C03626=1082.046,-23.655,-57.182,174.012,19.605,153.309
C03627=1082.052,-23.405,-57.194,174.013,19.607,153.309
C03628=1082.058,-23.155,-57.207,174.015,19.609,153.309
C03629=1082.064,-22.906,-57.220,174.016,19.611,153.310
C03630=1082.069,-22.656,-57.232,174.018,19.613,153.310
C03631=1082.075,-22.407,-57.246,174.019,19.615,153.310
C03632=1082.081,-22.157,-57.259,174.020,19.617,153.310
C03633=1082.087,-21.908,-57.272,174.022,19.619,153.310
C03634=1082.093,-21.658,-57.284,174.024,19.621,153.310
C03635=1082.099,-21.409,-57.298,174.025,19.623,153.310
C03636=1082.104,-21.158,-57.311,174.026,19.625,153.311
C03637=1082.110,-20.909,-57.324,174.028,19.627,153.311
C03638=1082.116,-20.659,-57.337,174.030,19.629,153.311
C03639=1082.122,-20.410,-57.350,174.031,19.631,153.311
C03640=1082.128,-20.160,-57.364,174.032,19.633,153.311
C03641=1082.134,-19.910,-57.376,174.034,19.635,153.311
C03642=1082.140,-19.661,-57.390,174.035,19.637,153.311
C03643=1082.146,-19.411,-57.402,174.037,19.639,153.311
C03644=1082.152,-19.162,-57.415,174.039,19.641,153.312
C03645=1082.157,-18.912,-57.429,174.040,19.643,153.312
C03646=1082.164,-18.663,-57.442,174.041,19.645,153.312
C03647=1082.170,-18.413,-57.455,174.042,19.647,153.312
C03648=1082.176,-18.163,-57.468,174.045,19.649,153.312
C03649=1082.181,-17.914,-57.482,174.046,19.651,153.312
C03650=1082.187,-17.664,-57.494,174.047,19.653,153.312
C03651=1082.194,-17.391,-57.509,174.048,19.655,153.313
C03652=1082.200,-17.116,-57.523,174.050,19.658,153.313
C03653=1082.206,-16.843,-57.538,174.052,19.660,153.313
C03654=1082.213,-16.568,-57.552,174.054,19.662,153.313
C03655=1082.220,-16.319,-57.565,174.055,19.664,153.313
C03656=1082.225,-16.069,-57.579,174.056,19.666,153.313
C03657=1082.231,-15.819,-57.592,174.058,19.668,153.313
C03658=1082.237,-15.570,-57.605,174.059,19.670,153.314
C03659=1082.243,-15.321,-57.618,174.061,19.672,153.314
C03660=1082.249,-15.071,-57.631,174.063,19.674,153.314
C03661=1082.255,-14.821,-57.645,174.064,19.676,153.314
C03662=1082.260,-14.572,-57.659,174.065,19.678,153.314
C03663=1082.266,-14.322,-57.671,174.066,19.680,153.314
C03664=1082.272,-14.073,-57.684,174.068,19.682,153.314
C03665=1082.278,-13.823,-57.698,174.070,19.684,153.314
C03666=1082.284,-13.574,-57.712,174.071,19.686,153.315
C03667=1082.289,-13.324,-57.725,174.072,19.688,153.315
C03668=1082.295,-13.074,-57.738,174.074,19.690,153.315
C03669=1082.301,-12.825,-57.752,174.076,19.692,153.315
C03670=1082.307,-12.576,-57.765,174.077,19.694,153.315
C03671=1082.312,-12.325,-57.778,174.078,19.696,153.315
C03672=1082.319,-12.076,-57.792,174.079,19.698,153.316
C03673=1082.324,-11.827,-57.805,174.082,19.700,153.316
C03674=1082.330,-11.577,-57.819,174.083,19.702,153.316
C03675=1082.336,-11.328,-57.833,174.084,19.704,153.316
C03676=1082.342,-11.078,-57.845,174.085,19.706,153.316
C03677=1082.348,-10.828,-57.859,174.087,19.708,153.316
C03678=1082.354,-10.578,-57.873,174.089,19.711,153.316
C03679=1082.360,-10.329,-57.886,174.090,19.713,153.317
C03680=1082.366,-10.079,-57.900,174.091,19.714,153.317
C03681=1082.372,-9.830,-57.913,174.093,19.716,153.317
C03682=1082.377,-9.580,-57.926,174.095,19.719,153.317
C03683=1082.383,-9.331,-57.939,174.096,19.721,153.317
C03684=1082.389,-9.081,-57.953,174.097,19.723,153.317
C03685=1082.395,-8.832,-57.967,174.099,19.725,153.318
C03686=1082.400,-8.582,-57.980,174.100,19.727,153.318
C03687=1082.407,-8.333,-57.994,174.102,19.729,153.318
C03688=1082.413,-8.083,-58.008,174.103,19.731,153.318
C03689=1082.418,-7.833,-58.022,174.105,19.733,153.318
C03690=1082.424,-7.584,-58.035,174.106,19.735,153.318
C03691=1082.430,-7.334,-58.048,174.108,19.738,153.318
C03692=1082.436,-7.084,-58.061,174.109,19.740,153.319
C03693=1082.441,-6.835,-58.075,174.110,19.742,153.319
C03694=1082.447,-6.586,-58.089,174.112,19.743,153.319
C03695=1082.454,-6.335,-58.103,174.113,19.745,153.319
C03696=1082.460,-6.086,-58.116,174.115,19.748,153.319
C03697=1082.465,-5.837,-58.130,174.117,19.750,153.319
C03698=1082.471,-5.587,-58.143,174.118,19.752,153.319
C03699=1082.477,-5.338,-58.157,174.119,19.754,153.320
C03700=1082.483,-5.088,-58.170,174.121,19.756,153.320
C03701=1082.489,-4.839,-58.184,174.123,19.758,153.320
C03702=1082.495,-4.589,-58.198,174.124,19.760,153.320
C03703=1082.501,-4.339,-58.212,174.125,19.762,153.320
C03704=1082.506,-4.090,-58.226,174.127,19.764,153.320
C03705=1082.513,-3.840,-58.239,174.128,19.766,153.320
C03706=1082.518,-3.591,-58.253,174.130,19.768,153.321
C03707=1082.525,-3.341,-58.266,174.131,19.770,153.321
C03708=1082.530,-3.091,-58.280,174.132,19.772,153.321
C03709=1082.536,-2.842,-58.294,174.134,19.775,153.321
C03710=1082.541,-2.592,-58.308,174.136,19.776,153.321
C03711=1082.548,-2.343,-58.321,174.137,19.778,153.321
C03712=1082.553,-2.094,-58.336,174.138,19.780,153.321
C03713=1082.559,-1.844,-58.350,174.140,19.783,153.322
C03714=1082.565,-1.594,-58.364,174.142,19.785,153.322
C03715=1082.571,-1.319,-58.379,174.143,19.787,153.322
C03716=1082.577,-1.043,-58.395,174.145,19.790,153.322
C03717=1082.584,-0.768,-58.409,174.146,19.792,153.322
C03718=1082.590,-0.492,-58.425,174.148,19.794,153.322
C03719=1082.596,-0.243,-58.439,174.149,19.796,153.323
C03720=1082.602,0.007,-58.452,174.151,19.798,153.323
C03721=1082.607,0.256,-58.466,174.153,19.801,153.323
C03722=1082.613,0.507,-58.480,174.154,19.803,153.323
C03723=1082.619,0.756,-58.494,174.155,19.805,153.323
C03724=1082.625,1.005,-58.508,174.156,19.807,153.323
C03725=1082.631,1.255,-58.522,174.158,19.809,153.324
C03726=1082.636,1.504,-58.536,174.160,19.811,153.324
C03727=1082.642,1.754,-58.550,174.161,19.813,153.324
C03728=1082.648,2.004,-58.564,174.162,19.815,153.324
C03729=1082.653,2.253,-58.579,174.164,19.818,153.324
C03730=1082.660,2.502,-58.592,174.166,19.820,153.324
C03731=1082.665,2.752,-58.606,174.167,19.821,153.324
C03732=1082.671,3.002,-58.620,174.168,19.823,153.325
C03733=1082.677,3.252,-58.634,174.170,19.826,153.325
C03734=1082.682,3.501,-58.649,174.172,19.828,153.325
C03735=1082.688,3.750,-58.662,174.173,19.830,153.325
C03736=1082.694,4.000,-58.677,174.174,19.832,153.325
C03737=1082.701,4.249,-58.691,174.176,19.834,153.325
C03738=1082.706,4.499,-58.704,174.178,19.836,153.326
C03739=1082.711,4.748,-58.718,174.179,19.838,153.326
C03740=1082.718,4.999,-58.733,174.180,19.840,153.326
C03741=1082.723,5.247,-58.747,174.182,19.843,153.326
C03742=1082.729,5.497,-58.761,174.183,19.845,153.326
C03743=1082.734,5.747,-58.775,174.185,19.847,153.326
C03744=1082.741,5.996,-58.790,174.186,19.849,153.327
C03745=1082.747,6.246,-58.803,174.188,19.851,153.327
C03746=1082.752,6.495,-58.817,174.189,19.853,153.327
C03747=1082.759,6.745,-58.832,174.190,19.855,153.327
C03748=1082.764,6.994,-58.846,174.192,19.857,153.327
C03749=1082.770,7.244,-58.860,174.194,19.859,153.327
C03750=1082.776,7.494,-58.875,174.195,19.861,153.327
C03751=1082.782,7.743,-58.888,174.197,19.863,153.328
C03752=1082.787,7.993,-58.902,174.199,19.866,153.328
C03753=1082.793,8.242,-58.917,174.200,19.868,153.328
C03754=1082.799,8.492,-58.931,174.201,19.870,153.328
C03755=1082.805,8.741,-58.945,174.202,19.872,153.328
C03756=1082.811,8.991,-58.959,174.205,19.874,153.328
C03757=1082.817,9.240,-58.974,174.206,19.876,153.329
C03758=1082.823,9.489,-58.988,174.207,19.878,153.329
C03759=1082.829,9.740,-59.002,174.208,19.880,153.329
C03760=1082.835,9.989,-59.017,174.210,19.883,153.329
C03761=1082.840,10.238,-59.030,174.212,19.884,153.329
C03762=1082.846,10.488,-59.045,174.213,19.886,153.329
C03763=1082.852,10.737,-59.059,174.214,19.888,153.330
C03764=1082.858,10.986,-59.074,174.217,19.891,153.330
C03765=1082.864,11.237,-59.088,174.218,19.893,153.330
C03766=1082.870,11.486,-59.103,174.219,19.895,153.330
C03767=1082.876,11.736,-59.117,174.221,19.897,153.330
C03768=1082.881,11.985,-59.131,174.222,19.899,153.330
C03769=1082.887,12.234,-59.145,174.224,19.902,153.330
C03770=1082.893,12.484,-59.160,174.225,19.904,153.331
C03771=1082.899,12.734,-59.174,174.227,19.906,153.331
C03772=1082.905,12.983,-59.189,174.228,19.907,153.331
C03773=1082.911,13.233,-59.203,174.230,19.909,153.331
C03774=1082.917,13.482,-59.217,174.231,19.911,153.331
C03775=1082.924,13.731,-59.232,174.233,19.914,153.331
C03776=1082.929,13.981,-59.246,174.234,19.916,153.332
C03777=1082.935,14.230,-59.261,174.236,19.918,153.332
C03778=1082.941,14.480,-59.275,174.238,19.920,153.332
C03779=1082.947,14.757,-59.291,174.239,19.922,153.332
C03780=1082.954,15.035,-59.307,174.241,19.925,153.332
C03781=1082.960,15.313,-59.323,174.242,19.927,153.332
C03782=1082.967,15.590,-59.339,174.244,19.930,153.333
C03783=1082.972,15.840,-59.354,174.245,19.932,153.333
C03784=1082.978,16.089,-59.369,174.247,19.934,153.333
C03785=1082.984,16.339,-59.384,174.249,19.936,153.333
C03786=1082.990,16.588,-59.398,174.250,19.938,153.333
C03787=1082.995,16.837,-59.412,174.252,19.940,153.333
C03788=1083.002,17.087,-59.427,174.253,19.942,153.333
C03789=1083.006,17.337,-59.442,174.255,19.944,153.334
C03790=1083.013,17.587,-59.457,174.256,19.946,153.334
C03791=1083.019,17.836,-59.471,174.257,19.948,153.334
C03792=1083.025,18.086,-59.485,174.260,19.951,153.334
C03793=1083.030,18.335,-59.500,174.261,19.953,153.334
C03794=1083.035,18.584,-59.515,174.262,19.955,153.334
C03795=1083.042,18.834,-59.529,174.263,19.957,153.335
C03796=1083.047,19.083,-59.544,174.265,19.959,153.335
C03797=1083.054,19.333,-59.559,174.267,19.961,153.335
C03798=1083.059,19.582,-59.574,174.268,19.963,153.335
C03799=1083.065,19.833,-59.588,174.270,19.966,153.335
C03800=1083.071,20.081,-59.603,174.271,19.968,153.335
C03801=1083.077,20.331,-59.618,174.273,19.970,153.336
C03802=1083.083,20.580,-59.632,174.275,19.972,153.336
C03803=1083.088,20.831,-59.647,174.276,19.974,153.336
C03804=1083.094,21.080,-59.662,174.277,19.976,153.336
C03805=1083.100,21.329,-59.676,174.278,19.978,153.336
C03806=1083.105,21.579,-59.692,174.281,19.981,153.336
C03807=1083.111,21.828,-59.707,174.282,19.983,153.337
C03808=1083.117,22.078,-59.721,174.283,19.985,153.337
C03809=1083.123,22.327,-59.735,174.285,19.987,153.337
C03810=1083.129,22.577,-59.751,174.286,19.989,153.337
C03811=1083.134,22.826,-59.765,174.288,19.991,153.337
C03812=1083.141,23.075,-59.780,174.290,19.993,153.337
C03813=1083.146,23.325,-59.796,174.291,19.995,153.337
C03814=1083.152,23.574,-59.811,174.293,19.997,153.338
C03815=1083.158,23.824,-59.824,174.294,19.999,153.338
C03816=1083.163,24.074,-59.840,174.296,20.002,153.338
C03817=1083.169,24.323,-59.855,174.297,20.004,153.338
C03818=1083.175,24.573,-59.870,174.298,20.006,153.338
C03819=1083.181,24.822,-59.885,174.301,20.008,153.338
C03820=1083.187,25.071,-59.900,174.302,20.010,153.339
C03821=1083.192,25.321,-59.915,174.303,20.012,153.339
C03822=1083.198,25.570,-59.930,174.305,20.015,153.339
C03823=1083.204,25.819,-59.944,174.306,20.017,153.339
C03824=1083.210,26.069,-59.960,174.308,20.019,153.339
C03825=1083.216,26.319,-59.975,174.310,20.021,153.339
C03826=1083.222,26.568,-59.989,174.311,20.023,153.340
C03827=1083.227,26.818,-60.004,174.312,20.025,153.340
C03828=1083.233,27.067,-60.019,174.315,20.028,153.340
C03829=1083.239,27.317,-60.034,174.316,20.030,153.340
C03830=1083.244,27.566,-60.049,174.317,20.031,153.340
C03831=1083.251,27.816,-60.064,174.319,20.033,153.340
C03832=1083.256,28.065,-60.079,174.321,20.036,153.340
C03833=1083.262,28.315,-60.094,174.322,20.038,153.341
C03834=1083.268,28.565,-60.109,174.323,20.040,153.341
C03835=1083.274,28.813,-60.125,174.325,20.042,153.341
C03836=1083.280,29.063,-60.140,174.327,20.044,153.341
C03837=1083.285,29.312,-60.155,174.328,20.046,153.341
C03838=1083.291,29.562,-60.170,174.330,20.049,153.341
C03839=1083.297,29.811,-60.185,174.331,20.051,153.342
C03840=1083.303,30.061,-60.201,174.332,20.053,153.342
C03841=1083.308,30.310,-60.215,174.335,20.055,153.342
C03842=1083.314,30.560,-60.231,174.336,20.057,153.342
C03843=1083.321,30.839,-60.247,174.338,20.060,153.342
C03844=1083.327,31.118,-60.265,174.339,20.062,153.342
C03845=1083.333,31.397,-60.281,174.341,20.065,153.343
C03846=1083.340,31.676,-60.299,174.342,20.067,153.343
C03847=1083.345,31.925,-60.313,174.344,20.069,153.343
C03848=1083.351,32.175,-60.330,174.346,20.071,153.343
C03849=1083.357,32.424,-60.344,174.347,20.073,153.343
C03850=1083.363,32.674,-60.360,174.349,20.076,153.343
C03851=1083.368,32.924,-60.375,174.351,20.077,153.343
C03852=1083.374,33.173,-60.390,174.352,20.079,153.344
C03853=1083.380,33.422,-60.405,174.354,20.082,153.344
C03854=1083.386,33.672,-60.420,174.355,20.084,153.344
C03855=1083.392,33.921,-60.436,174.357,20.086,153.344
C03856=1083.397,34.171,-60.452,174.359,20.088,153.344
C03857=1083.403,34.420,-60.466,174.360,20.090,153.344
C03858=1083.409,34.670,-60.482,174.361,20.092,153.345
C03859=1083.415,34.919,-60.498,174.363,20.095,153.345
C03860=1083.420,35.168,-60.513,174.365,20.097,153.345
C03861=1083.426,35.418,-60.528,174.366,20.099,153.345
C03862=1083.432,35.668,-60.543,174.368,20.101,153.345
C03863=1083.437,35.917,-60.558,174.369,20.103,153.345
C03864=1083.444,36.166,-60.574,174.371,20.105,153.345
C03865=1083.450,36.416,-60.590,174.373,20.107,153.346
C03866=1083.455,36.665,-60.605,174.374,20.109,153.346
C03867=1083.462,36.914,-60.620,174.375,20.111,153.346
C03868=1083.467,37.164,-60.636,174.377,20.113,153.346
C03869=1083.472,37.413,-60.651,174.379,20.115,153.346
C03870=1083.479,37.662,-60.667,174.380,20.117,153.346
C03871=1083.485,37.912,-60.682,174.382,20.120,153.347
C03872=1083.490,38.162,-60.698,174.383,20.122,153.347
C03873=1083.496,38.411,-60.712,174.385,20.124,153.347
C03874=1083.502,38.661,-60.729,174.387,20.126,153.347
C03875=1083.508,38.911,-60.744,174.388,20.128,153.347
C03876=1083.513,39.159,-60.760,174.390,20.131,153.347
C03877=1083.519,39.409,-60.776,174.392,20.132,153.347
C03878=1083.525,39.659,-60.791,174.393,20.134,153.348
C03879=1083.530,39.908,-60.806,174.395,20.137,153.348
C03880=1083.536,40.158,-60.822,174.396,20.139,153.348
C03881=1083.542,40.408,-60.838,174.398,20.141,153.348
C03882=1083.547,40.656,-60.853,174.400,20.143,153.348
C03883=1083.553,40.906,-60.868,174.401,20.145,153.348
C03884=1083.559,41.155,-60.885,174.402,20.147,153.349
C03885=1083.564,41.404,-60.900,174.404,20.150,153.349
C03886=1083.570,41.654,-60.916,174.406,20.152,153.349
C03887=1083.576,41.904,-60.932,174.407,20.154,153.349
C03888=1083.582,42.153,-60.947,174.409,20.156,153.349
C03889=1083.588,42.402,-60.962,174.410,20.158,153.349
C03890=1083.593,42.652,-60.978,174.412,20.161,153.350
C03891=1083.599,42.901,-60.994,174.414,20.162,153.350
C03892=1083.605,43.151,-61.010,174.415,20.164,153.350
C03893=1083.610,43.400,-61.026,174.417,20.167,153.350
C03894=1083.617,43.650,-61.041,174.419,20.169,153.350
C03895=1083.623,43.899,-61.057,174.420,20.171,153.350
C03896=1083.628,44.149,-61.072,174.422,20.173,153.350
C03897=1083.634,44.398,-61.088,174.423,20.175,153.351
C03898=1083.639,44.648,-61.104,174.424,20.177,153.351
C03899=1083.645,44.897,-61.120,174.427,20.180,153.351
C03900=1083.650,45.146,-61.135,174.428,20.182,153.351
C03901=1083.656,45.396,-61.152,174.430,20.184,153.351
C03902=1083.662,45.645,-61.168,174.431,20.186,153.351
C03903=1083.668,45.895,-61.183,174.433,20.188,153.352
C03904=1083.673,46.144,-61.199,174.435,20.190,153.352
C03905=1083.678,46.394,-61.215,174.436,20.192,153.352
C03906=1083.684,46.643,-61.232,174.437,20.194,153.352
C03907=1083.690,46.923,-61.249,174.439,20.197,153.352
C03908=1083.697,47.201,-61.267,174.441,20.199,153.352
C03909=1083.703,47.480,-61.285,174.443,20.201,153.353
C03910=1083.709,47.759,-61.302,174.445,20.204,153.353
C03911=1083.715,48.008,-61.319,174.446,20.206,153.353
C03912=1083.721,48.258,-61.335,174.448,20.208,153.353
C03913=1083.726,48.508,-61.350,174.450,20.210,153.353
C03914=1083.732,48.756,-61.366,174.452,20.213,153.353
C03915=1083.738,49.006,-61.382,174.453,20.215,153.353
C03916=1083.743,49.256,-61.398,174.454,20.217,153.354
C03917=1083.749,49.505,-61.414,174.456,20.219,153.354
C03918=1083.755,49.754,-61.431,174.458,20.221,153.354
C03919=1083.760,50.004,-61.446,174.460,20.224,153.354
C03920=1083.766,50.253,-61.462,174.461,20.225,153.354
C03921=1083.772,50.502,-61.478,174.462,20.227,153.354
C03922=1083.778,50.752,-61.494,174.465,20.230,153.354
C03923=1083.783,51.002,-61.511,174.466,20.232,153.355
C03924=1083.789,51.251,-61.527,174.467,20.234,153.355
C03925=1083.794,51.500,-61.543,174.469,20.236,153.355
C03926=1083.800,51.749,-61.559,174.471,20.238,153.355
C03927=1083.806,51.999,-61.575,174.473,20.240,153.355
C03928=1083.812,52.249,-61.591,174.474,20.242,153.355
C03929=1083.818,52.498,-61.607,174.475,20.244,153.356
C03930=1083.824,52.747,-61.623,174.478,20.246,153.356
C03931=1083.829,52.997,-61.639,174.479,20.248,153.356
C03932=1083.834,53.246,-61.655,174.481,20.251,153.356
C03933=1083.840,53.496,-61.672,174.482,20.253,153.356
C03934=1083.846,53.745,-61.688,174.484,20.255,153.356
C03935=1083.852,53.994,-61.704,174.486,20.257,153.356
C03936=1083.858,54.244,-61.720,174.487,20.259,153.356
C03937=1083.863,54.494,-61.736,174.489,20.261,153.357
C03938=1083.869,54.743,-61.752,174.491,20.263,153.357
C03939=1083.875,54.992,-61.768,174.492,20.265,153.357
C03940=1083.880,55.241,-61.785,174.494,20.268,153.357
C03941=1083.886,55.491,-61.801,174.495,20.269,153.357
C03942=1083.892,55.740,-61.817,174.498,20.272,153.357
C03943=1083.898,55.989,-61.834,174.499,20.274,153.357
C03944=1083.904,56.239,-61.850,174.500,20.276,153.358
C03945=1083.910,56.488,-61.866,174.502,20.278,153.358
C03946=1083.915,56.738,-61.882,174.504,20.280,153.358
C03947=1083.921,56.988,-61.899,174.506,20.282,153.358
C03948=1083.927,57.237,-61.915,174.507,20.284,153.358
C03949=1083.932,57.486,-61.931,174.508,20.286,153.358
C03950=1083.938,57.736,-61.947,174.511,20.288,153.358
C03951=1083.944,57.985,-61.964,174.512,20.290,153.359
C03952=1083.950,58.235,-61.980,174.514,20.292,153.359
C03953=1083.956,58.484,-61.997,174.516,20.294,153.359
C03954=1083.962,58.733,-62.013,174.517,20.296,153.359
C03955=1083.967,58.983,-62.029,174.519,20.298,153.359
C03956=1083.973,59.232,-62.046,174.520,20.300,153.359
C03957=1083.979,59.482,-62.062,174.523,20.303,153.359
C03958=1083.985,59.731,-62.079,174.524,20.305,153.360
C03959=1083.991,59.980,-62.095,174.525,20.306,153.360
C03960=1083.996,60.230,-62.111,174.527,20.309,153.360
C03961=1084.002,60.479,-62.128,174.529,20.311,153.360
C03962=1084.008,60.729,-62.144,174.531,20.313,153.360
C03963=1084.014,60.977,-62.161,174.532,20.315,153.360
C03964=1084.020,61.227,-62.177,174.534,20.317,153.360
C03965=1084.026,61.476,-62.194,174.536,20.319,153.360
C03966=1084.031,61.726,-62.211,174.537,20.321,153.360
C03967=1084.037,61.975,-62.227,174.539,20.323,153.361
C03968=1084.043,62.225,-62.243,174.541,20.325,153.361
C03969=1084.049,62.474,-62.259,174.543,20.327,153.361
C03970=1084.054,62.724,-62.276,174.544,20.329,153.361
C03971=1084.061,63.002,-62.295,174.546,20.331,153.361
C03972=1084.067,63.281,-62.313,174.548,20.333,153.361
C03973=1084.074,63.559,-62.331,174.550,20.336,153.361
C03974=1084.080,63.838,-62.349,174.552,20.338,153.362
C03975=1084.087,64.088,-62.367,174.554,20.340,153.362
C03976=1084.093,64.337,-62.384,174.556,20.342,153.362
C03977=1084.098,64.587,-62.400,174.557,20.344,153.362
C03978=1084.104,64.836,-62.417,174.558,20.346,153.362
C03979=1084.110,65.086,-62.433,174.561,20.348,153.362
C03980=1084.115,65.335,-62.450,174.562,20.350,153.362
C03981=1084.121,65.584,-62.467,174.564,20.353,153.362
C03982=1084.127,65.833,-62.483,174.565,20.354,153.362
C03983=1084.132,66.083,-62.500,174.568,20.356,153.363
C03984=1084.139,66.332,-62.517,174.569,20.358,153.363
C03985=1084.144,66.581,-62.534,174.571,20.361,153.363
C03986=1084.150,66.831,-62.550,174.573,20.362,153.363
C03987=1084.155,67.080,-62.567,174.574,20.364,153.363
C03988=1084.161,67.329,-62.584,174.576,20.367,153.363
C03989=1084.166,67.579,-62.601,174.577,20.369,153.363
C03990=1084.172,67.828,-62.617,174.580,20.371,153.363
C03991=1084.178,68.078,-62.634,174.581,20.373,153.364
C03992=1084.184,68.327,-62.651,174.583,20.375,153.364
C03993=1084.190,68.577,-62.668,174.585,20.377,153.364
C03994=1084.196,68.826,-62.684,174.586,20.379,153.364
C03995=1084.201,69.075,-62.702,174.588,20.381,153.364
C03996=1084.207,69.325,-62.718,174.589,20.383,153.364
C03997=1084.212,69.574,-62.735,174.592,20.385,153.364
C03998=1084.218,69.823,-62.752,174.593,20.387,153.364
C03999=1084.224,70.073,-62.769,174.595,20.389,153.365
C04000=1084.229,70.322,-62.786,174.596,20.391,153.365
C04001=1084.235,70.571,-62.802,174.599,20.393,153.365
C04002=1084.240,70.821,-62.819,174.600,20.395,153.365
C04003=1084.247,71.070,-62.837,174.601,20.397,153.365
C04004=1084.252,71.320,-62.854,174.604,20.399,153.365
C04005=1084.258,71.569,-62.871,174.605,20.401,153.365
C04006=1084.264,71.818,-62.887,174.607,20.404,153.365
C04007=1084.269,72.068,-62.904,174.608,20.405,153.366
C04008=1084.275,72.317,-62.922,174.611,20.408,153.366
C04009=1084.281,72.566,-62.938,174.612,20.410,153.366
C04010=1084.286,72.815,-62.956,174.614,20.412,153.366
C04011=1084.291,73.065,-62.972,174.616,20.414,153.366
C04012=1084.298,73.314,-62.990,174.618,20.416,153.366
C04013=1084.303,73.564,-63.007,174.619,20.417,153.366
C04014=1084.309,73.813,-63.024,174.620,20.419,153.366
C04015=1084.315,74.063,-63.040,174.623,20.422,153.367
C04016=1084.320,74.312,-63.058,174.624,20.423,153.367
C04017=1084.326,74.561,-63.075,174.626,20.426,153.367
C04018=1084.332,74.811,-63.092,174.628,20.428,153.367
C04019=1084.338,75.060,-63.109,174.630,20.430,153.367
C04020=1084.343,75.309,-63.127,174.631,20.432,153.367
C04021=1084.349,75.559,-63.143,174.633,20.434,153.367
C04022=1084.355,75.808,-63.160,174.635,20.436,153.367
C04023=1084.360,76.057,-63.178,174.637,20.438,153.367
C04024=1084.367,76.307,-63.195,174.638,20.440,153.368
C04025=1084.372,76.556,-63.212,174.641,20.442,153.368
C04026=1084.377,76.806,-63.229,174.642,20.444,153.368
C04027=1084.383,77.055,-63.247,174.643,20.445,153.368
C04028=1084.389,77.303,-63.264,174.646,20.448,153.368
C04029=1084.395,77.554,-63.281,174.647,20.450,153.368
C04030=1084.401,77.803,-63.298,174.649,20.452,153.368
C04031=1084.406,78.052,-63.315,174.650,20.454,153.368
C04032=1084.412,78.301,-63.332,174.653,20.456,153.368
C04033=1084.418,78.550,-63.350,174.654,20.458,153.368
C04034=1084.423,78.800,-63.367,174.656,20.460,153.369
C04035=1084.429,79.079,-63.386,174.658,20.463,153.369
C04036=1084.436,79.358,-63.406,174.660,20.464,153.369
C04037=1084.442,79.636,-63.425,174.662,20.467,153.369
C04038=1084.448,79.915,-63.445,174.664,20.469,153.369
C04039=1084.455,80.164,-63.462,174.665,20.471,153.369
C04040=1084.460,80.413,-63.480,174.668,20.473,153.369
C04041=1084.465,80.663,-63.496,174.669,20.475,153.369
C04042=1084.471,80.912,-63.514,174.671,20.477,153.370
C04043=1084.477,81.161,-63.532,174.673,20.479,153.370
C04044=1084.482,81.411,-63.549,174.675,20.481,153.370
C04045=1084.488,81.660,-63.566,174.676,20.483,153.370
C04046=1084.493,81.909,-63.584,174.679,20.485,153.370
C04047=1084.499,82.159,-63.602,174.680,20.487,153.370
C04048=1084.505,82.408,-63.619,174.682,20.489,153.370
C04049=1084.510,82.658,-63.636,174.684,20.491,153.370
C04050=1084.516,82.907,-63.654,174.686,20.493,153.370
C04051=1084.522,83.156,-63.672,174.687,20.495,153.371
C04052=1084.527,83.405,-63.689,174.689,20.497,153.371
C04053=1084.533,83.654,-63.706,174.691,20.499,153.371
C04054=1084.539,83.904,-63.723,174.693,20.501,153.371
C04055=1084.545,84.154,-63.741,174.694,20.503,153.371
C04056=1084.550,84.403,-63.759,174.697,20.505,153.371
C04057=1084.556,84.652,-63.776,174.698,20.507,153.371
C04058=1084.562,84.901,-63.794,174.700,20.509,153.371
C04059=1084.567,85.150,-63.812,174.702,20.511,153.371
C04060=1084.573,85.400,-63.829,174.704,20.513,153.371
C04061=1084.579,85.649,-63.847,174.705,20.515,153.372
C04062=1084.585,85.898,-63.865,174.708,20.517,153.372
C04063=1084.590,86.148,-63.882,174.709,20.519,153.372
C04064=1084.596,86.398,-63.900,174.711,20.521,153.372
C04065=1084.601,86.647,-63.917,174.713,20.523,153.372
C04066=1084.607,86.896,-63.935,174.715,20.525,153.372
C04067=1084.613,87.146,-63.953,174.716,20.527,153.372
C04068=1084.619,87.395,-63.970,174.719,20.529,153.372
C04069=1084.624,87.644,-63.988,174.720,20.531,153.372
C04070=1084.630,87.893,-64.006,174.722,20.533,153.372
C04071=1084.636,88.142,-64.023,174.724,20.535,153.373
C04072=1084.641,88.391,-64.041,174.726,20.537,153.373
C04073=1084.647,88.641,-64.059,174.727,20.538,153.373
C04074=1084.653,88.890,-64.076,174.730,20.540,153.373
C04075=1084.658,89.139,-64.094,174.731,20.542,153.373
C04076=1084.665,89.389,-64.112,174.733,20.544,153.373
C04077=1084.670,89.638,-64.129,174.735,20.546,153.373
C04078=1084.676,89.888,-64.147,174.737,20.548,153.373
C04079=1084.681,90.137,-64.165,174.738,20.550,153.373
C04080=1084.686,90.386,-64.183,174.741,20.552,153.373
C04081=1084.693,90.636,-64.201,174.742,20.554,153.373
C04082=1084.698,90.884,-64.219,174.744,20.556,153.373
C04083=1084.705,91.134,-64.237,174.746,20.558,153.373
C04084=1084.710,91.383,-64.255,174.748,20.560,153.374
C04085=1084.716,91.632,-64.272,174.749,20.561,153.374
C04086=1084.721,91.882,-64.291,174.751,20.564,153.374
C04087=1084.727,92.131,-64.308,174.753,20.565,153.374
C04088=1084.732,92.380,-64.326,174.755,20.568,153.374
C04089=1084.738,92.630,-64.344,174.757,20.569,153.374
C04090=1084.744,92.879,-64.362,174.759,20.572,153.374
C04091=1084.749,93.128,-64.381,174.760,20.573,153.374
C04092=1084.755,93.378,-64.398,174.762,20.576,153.374
C04093=1084.760,93.627,-64.416,174.765,20.577,153.374
C04094=1084.767,93.876,-64.434,174.766,20.579,153.375
C04095=1084.771,94.126,-64.452,174.768,20.581,153.375
C04096=1084.778,94.375,-64.471,174.770,20.583,153.375
C04097=1084.783,94.624,-64.488,174.772,20.585,153.375
C04098=1084.788,94.873,-64.506,174.774,20.587,153.375
C04099=1084.795,95.152,-64.526,174.776,20.589,153.375
C04100=1084.802,95.431,-64.547,174.778,20.592,153.375
C04101=1084.807,95.710,-64.567,174.780,20.594,153.375
C04102=1084.814,95.988,-64.587,174.782,20.596,153.375
C04103=1084.820,96.237,-64.605,174.784,20.597,153.375
C04104=1084.825,96.488,-64.623,174.786,20.600,153.375
C04105=1084.831,96.736,-64.642,174.788,20.601,153.375
C04106=1084.837,96.986,-64.659,174.790,20.603,153.375
C04107=1084.842,97.235,-64.677,174.791,20.605,153.376
C04108=1084.848,97.484,-64.696,174.794,20.607,153.376
C04109=1084.854,97.733,-64.714,174.795,20.609,153.376
C04110=1084.860,97.983,-64.732,174.797,20.611,153.376
C04111=1084.865,98.232,-64.751,174.799,20.613,153.376
C04112=1084.871,98.481,-64.769,174.801,20.615,153.376
C04113=1084.876,98.730,-64.786,174.803,20.616,153.376
C04114=1084.882,98.980,-64.805,174.805,20.618,153.376
C04115=1084.888,99.229,-64.823,174.807,20.621,153.376
C04116=1084.894,99.478,-64.842,174.809,20.622,153.376
C04117=1084.899,99.727,-64.860,174.811,20.624,153.376
C04118=1084.905,99.977,-64.878,174.812,20.626,153.376
C04119=1084.911,100.226,-64.896,174.815,20.628,153.376
C04120=1084.916,100.476,-64.915,174.816,20.630,153.377
C04121=1084.922,100.724,-64.933,174.818,20.632,153.377
C04122=1084.928,100.974,-64.951,174.820,20.633,153.377
C04123=1084.933,101.223,-64.969,174.822,20.635,153.377
C04124=1084.939,101.472,-64.988,174.824,20.638,153.377
C04125=1084.944,101.722,-65.006,174.826,20.639,153.377
C04126=1084.951,101.971,-65.024,174.828,20.641,153.377
C04127=1084.955,102.220,-65.043,174.830,20.643,153.377
C04128=1084.962,102.469,-65.061,174.832,20.645,153.377
C04129=1084.967,102.719,-65.079,174.833,20.647,153.377
C04130=1084.973,102.968,-65.098,174.836,20.649,153.377
C04131=1084.978,103.218,-65.117,174.838,20.651,153.377
C04132=1084.984,103.466,-65.135,174.839,20.652,153.377
C04133=1084.990,103.716,-65.153,174.842,20.655,153.377
C04134=1084.995,103.965,-65.172,174.843,20.656,153.378
C04135=1085.001,104.214,-65.191,174.845,20.659,153.378
C04136=1085.006,104.463,-65.209,174.847,20.660,153.378
C04137=1085.012,104.713,-65.228,174.849,20.662,153.378
C04138=1085.017,104.962,-65.246,174.852,20.664,153.378
C04139=1085.023,105.211,-65.264,174.853,20.666,153.378
C04140=1085.029,105.461,-65.283,174.855,20.668,153.378
C04141=1085.034,105.710,-65.302,174.857,20.669,153.378
C04142=1085.040,105.959,-65.321,174.859,20.672,153.378
C04143=1085.045,106.208,-65.339,174.860,20.673,153.378
C04144=1085.052,106.457,-65.357,174.863,20.675,153.378
C04145=1085.057,106.706,-65.376,174.865,20.678,153.378
C04146=1085.063,106.956,-65.394,174.866,20.679,153.378
C04147=1085.068,107.205,-65.413,174.869,20.681,153.378
C04148=1085.074,107.454,-65.432,174.870,20.682,153.378
C04149=1085.080,107.704,-65.450,174.872,20.685,153.379
C04150=1085.085,107.953,-65.469,174.874,20.686,153.379
C04151=1085.091,108.202,-65.488,174.876,20.688,153.379
C04152=1085.097,108.452,-65.506,174.879,20.690,153.379
C04153=1085.102,108.700,-65.525,174.880,20.692,153.379
C04154=1085.108,108.950,-65.544,174.882,20.694,153.379
C04155=1085.113,109.200,-65.562,174.884,20.696,153.379
C04156=1085.119,109.448,-65.581,174.886,20.698,153.379
C04157=1085.125,109.697,-65.600,174.889,20.699,153.379
C04158=1085.131,109.947,-65.619,174.890,20.701,153.379
C04159=1085.136,110.195,-65.637,174.892,20.703,153.379
C04160=1085.142,110.445,-65.656,174.894,20.705,153.379
C04161=1085.148,110.695,-65.675,174.896,20.707,153.379
C04162=1085.153,110.943,-65.693,174.899,20.709,153.379
C04163=1085.160,111.222,-65.715,174.900,20.711,153.379
C04164=1085.166,111.501,-65.736,174.902,20.713,153.379
C04165=1085.172,111.780,-65.757,174.905,20.714,153.379
C04166=1085.178,112.059,-65.778,174.907,20.717,153.379
C04167=1085.184,112.308,-65.797,174.909,20.719,153.379
C04168=1085.190,112.557,-65.816,174.911,20.720,153.379
C04169=1085.196,112.806,-65.835,174.913,20.722,153.379
C04170=1085.201,113.056,-65.854,174.915,20.724,153.380
C04171=1085.207,113.306,-65.872,174.917,20.726,153.380
C04172=1085.212,113.554,-65.891,174.919,20.728,153.380
C04173=1085.218,113.803,-65.910,174.921,20.729,153.380
C04174=1085.224,114.053,-65.929,174.923,20.731,153.380
C04175=1085.229,114.302,-65.948,174.925,20.733,153.380
C04176=1085.235,114.551,-65.967,174.927,20.735,153.380
C04177=1085.241,114.800,-65.986,174.929,20.737,153.380
C04178=1085.247,115.050,-66.005,174.931,20.739,153.380
C04179=1085.252,115.298,-66.024,174.933,20.741,153.380
C04180=1085.257,115.548,-66.043,174.935,20.742,153.380
C04181=1085.263,115.797,-66.062,174.937,20.744,153.380
C04182=1085.268,116.046,-66.081,174.939,20.746,153.380
C04183=1085.274,116.295,-66.101,174.941,20.748,153.380
C04184=1085.280,116.545,-66.120,174.943,20.750,153.380
C04185=1085.285,116.794,-66.139,174.945,20.752,153.380
C04186=1085.290,117.043,-66.158,174.947,20.754,153.380
C04187=1085.296,117.292,-66.177,174.949,20.756,153.380
C04188=1085.302,117.542,-66.196,174.951,20.757,153.380
C04189=1085.307,117.791,-66.215,174.953,20.759,153.381
C04190=1085.313,118.040,-66.235,174.955,20.761,153.381
C04191=1085.318,118.289,-66.254,174.957,20.763,153.381
C04192=1085.323,118.538,-66.273,174.959,20.765,153.381
C04193=1085.329,118.788,-66.292,174.961,20.767,153.381
C04194=1085.335,119.037,-66.311,174.964,20.769,153.381
C04195=1085.340,119.286,-66.330,174.965,20.770,153.381
C04196=1085.345,119.535,-66.349,174.968,20.772,153.381
C04197=1085.351,119.784,-66.369,174.970,20.774,153.381
C04198=1085.357,120.033,-66.389,174.971,20.776,153.381
C04199=1085.363,120.283,-66.408,174.974,20.778,153.381
C04200=1085.368,120.532,-66.427,174.975,20.779,153.381
C04201=1085.374,120.781,-66.446,174.978,20.781,153.381
C04202=1085.379,121.030,-66.465,174.980,20.783,153.381
C04203=1085.385,121.280,-66.484,174.981,20.784,153.381
C04204=1085.391,121.529,-66.504,174.984,20.786,153.381
C04205=1085.396,121.777,-66.523,174.986,20.788,153.381
C04206=1085.402,122.027,-66.542,174.988,20.790,153.381
C04207=1085.407,122.276,-66.562,174.990,20.792,153.381
C04208=1085.413,122.525,-66.582,174.992,20.794,153.381
C04209=1085.419,122.775,-66.601,174.994,20.796,153.381
C04210=1085.424,123.024,-66.621,174.996,20.797,153.381
C04211=1085.429,123.273,-66.640,174.999,20.799,153.381
C04212=1085.435,123.522,-66.660,175.000,20.801,153.381
C04213=1085.441,123.771,-66.679,175.002,20.803,153.381
C04214=1085.447,124.021,-66.698,175.005,20.805,153.381
C04215=1085.452,124.270,-66.717,175.006,20.806,153.382
C04216=1085.458,124.519,-66.737,175.009,20.808,153.382
C04217=1085.464,124.768,-66.756,175.011,20.810,153.382
C04218=1085.469,125.017,-66.775,175.013,20.811,153.382
C04219=1085.475,125.266,-66.795,175.015,20.813,153.382
C04220=1085.481,125.515,-66.815,175.017,20.815,153.382
C04221=1085.486,125.765,-66.834,175.019,20.817,153.382
C04222=1085.492,126.014,-66.854,175.021,20.819,153.382
C04223=1085.497,126.263,-66.874,175.024,20.821,153.382
C04224=1085.503,126.513,-66.893,175.025,20.822,153.382
C04225=1085.509,126.762,-66.913,175.028,20.824,153.382
C04226=1085.515,127.011,-66.932,175.030,20.826,153.382
C04227=1085.521,127.289,-66.954,175.032,20.828,153.382
C04228=1085.527,127.568,-66.976,175.034,20.829,153.382
C04229=1085.533,127.847,-66.997,175.036,20.831,153.382
C04230=1085.540,128.126,-67.020,175.039,20.833,153.382
C04231=1085.545,128.376,-67.039,175.041,20.835,153.382
C04232=1085.551,128.624,-67.059,175.043,20.837,153.382
C04233=1085.557,128.874,-67.079,175.046,20.839,153.382
C04234=1085.563,129.123,-67.099,175.047,20.840,153.382
C04235=1085.568,129.371,-67.117,175.050,20.842,153.382
C04236=1085.574,129.620,-67.137,175.052,20.844,153.382
C04237=1085.579,129.870,-67.157,175.054,20.845,153.382
C04238=1085.585,130.119,-67.177,175.056,20.847,153.382
C04239=1085.591,130.368,-67.196,175.059,20.849,153.382
C04240=1085.597,130.617,-67.216,175.060,20.850,153.382
C04241=1085.602,130.866,-67.236,175.062,20.852,153.382
C04242=1085.608,131.115,-67.256,175.065,20.854,153.382
C04243=1085.614,131.364,-67.276,175.067,20.855,153.382
C04244=1085.619,131.614,-67.295,175.069,20.857,153.382
C04245=1085.625,131.863,-67.315,175.071,20.859,153.382
C04246=1085.631,132.112,-67.335,175.073,20.860,153.382
C04247=1085.636,132.361,-67.355,175.075,20.862,153.382
C04248=1085.642,132.611,-67.374,175.078,20.864,153.382
C04249=1085.648,132.859,-67.394,175.080,20.866,153.382
C04250=1085.653,133.109,-67.415,175.082,20.868,153.382
C04251=1085.659,133.358,-67.434,175.084,20.870,153.382
C04252=1085.665,133.607,-67.454,175.087,20.871,153.382
C04253=1085.670,133.856,-67.475,175.088,20.872,153.382
C04254=1085.676,134.105,-67.494,175.090,20.874,153.382
C04255=1085.681,134.354,-67.514,175.093,20.876,153.382
C04256=1085.687,134.603,-67.534,175.094,20.878,153.382
C04257=1085.693,134.853,-67.554,175.097,20.880,153.382
C04258=1085.698,135.102,-67.574,175.099,20.881,153.382
C04259=1085.704,135.351,-67.594,175.101,20.883,153.382
C04260=1085.709,135.600,-67.614,175.103,20.885,153.382
C04261=1085.715,135.849,-67.634,175.106,20.886,153.382
C04262=1085.720,136.098,-67.655,175.108,20.888,153.382
C04263=1085.726,136.347,-67.674,175.110,20.890,153.382
C04264=1085.732,136.597,-67.694,175.112,20.892,153.382
C04265=1085.738,136.846,-67.715,175.114,20.893,153.382
C04266=1085.744,137.095,-67.735,175.117,20.895,153.382
C04267=1085.749,137.344,-67.755,175.118,20.897,153.382
C04268=1085.755,137.593,-67.775,175.121,20.898,153.382
C04269=1085.760,137.843,-67.795,175.123,20.900,153.382
C04270=1085.766,138.092,-67.815,175.126,20.902,153.382
C04271=1085.771,138.341,-67.835,175.127,20.903,153.382
C04272=1085.777,138.590,-67.855,175.129,20.905,153.382
C04273=1085.783,138.839,-67.876,175.132,20.907,153.382
C04274=1085.789,139.088,-67.896,175.134,20.908,153.382
C04275=1085.793,139.337,-67.916,175.136,20.910,153.382
C04276=1085.799,139.586,-67.936,175.138,20.912,153.382
C04277=1085.805,139.835,-67.956,175.141,20.914,153.382
C04278=1085.811,140.085,-67.977,175.142,20.915,153.382
C04279=1085.817,140.334,-67.997,175.145,20.917,153.382
C04280=1085.823,140.583,-68.017,175.147,20.919,153.382
C04281=1085.828,140.832,-68.038,175.150,20.921,153.382
C04282=1085.833,141.081,-68.058,175.151,20.922,153.382
C04283=1085.839,141.330,-68.078,175.154,20.924,153.382
C04284=1085.844,141.579,-68.099,175.156,20.925,153.382
C04285=1085.850,141.828,-68.119,175.159,20.927,153.382
C04286=1085.856,142.077,-68.139,175.160,20.929,153.382
C04287=1085.861,142.327,-68.159,175.162,20.931,153.382
C04288=1085.866,142.576,-68.180,175.165,20.933,153.382
C04289=1085.872,142.825,-68.200,175.167,20.934,153.382
C04290=1085.878,143.074,-68.221,175.169,20.936,153.382
C04291=1085.884,143.352,-68.244,175.171,20.937,153.382
C04292=1085.890,143.632,-68.266,175.175,20.940,153.382
C04293=1085.896,143.910,-68.290,175.177,20.942,153.382
C04294=1085.903,144.189,-68.312,175.179,20.944,153.382
C04295=1085.909,144.438,-68.332,175.182,20.945,153.382
C04296=1085.914,144.687,-68.353,175.183,20.946,153.382
C04297=1085.919,144.936,-68.373,175.186,20.948,153.382
C04298=1085.924,145.185,-68.394,175.188,20.950,153.382
C04299=1085.931,145.433,-68.415,175.191,20.952,153.382
C04300=1085.937,145.683,-68.436,175.192,20.953,153.382
C04301=1085.942,145.932,-68.456,175.195,20.955,153.382
C04302=1085.948,146.181,-68.476,175.197,20.956,153.382
C04303=1085.953,146.430,-68.497,175.200,20.958,153.382
C04304=1085.958,146.679,-68.517,175.201,20.960,153.382
C04305=1085.965,146.929,-68.537,175.204,20.961,153.382
C04306=1085.971,147.177,-68.559,175.206,20.963,153.382
C04307=1085.976,147.426,-68.579,175.209,20.965,153.382
C04308=1085.981,147.676,-68.600,175.211,20.966,153.381
C04309=1085.988,147.925,-68.620,175.213,20.968,153.382
C04310=1085.993,148.174,-68.641,175.215,20.970,153.382
C04311=1085.998,148.423,-68.662,175.218,20.971,153.381
C04312=1086.004,148.672,-68.683,175.220,20.973,153.381
C04313=1086.009,148.921,-68.703,175.222,20.975,153.381
C04314=1086.015,149.171,-68.724,175.224,20.977,153.381
C04315=1086.021,149.419,-68.745,175.227,20.978,153.381
C04316=1086.026,149.668,-68.765,175.229,20.980,153.381
C04317=1086.032,149.917,-68.786,175.231,20.982,153.381
C04318=1086.037,150.167,-68.807,175.233,20.983,153.381
C04319=1086.043,150.416,-68.828,175.236,20.985,153.381
C04320=1086.048,150.665,-68.849,175.238,20.987,153.381
C04321=1086.054,150.914,-68.869,175.241,20.988,153.381
C04322=1086.060,151.163,-68.891,175.243,20.990,153.381
C04323=1086.066,151.412,-68.911,175.244,20.991,153.381
C04324=1086.071,151.661,-68.931,175.247,20.993,153.381
C04325=1086.077,151.909,-68.953,175.249,20.995,153.381
C04326=1086.082,152.159,-68.973,175.252,20.996,153.381
C04327=1086.088,152.408,-68.994,175.254,20.998,153.381
C04328=1086.093,152.657,-69.015,175.256,20.999,153.381
C04329=1086.098,152.906,-69.036,175.258,21.001,153.381
C04330=1086.105,153.155,-69.057,175.261,21.003,153.381
C04331=1086.110,153.404,-69.078,175.263,21.005,153.381
C04332=1086.115,153.654,-69.099,175.266,21.006,153.381
C04333=1086.121,153.903,-69.120,175.267,21.007,153.381
C04334=1086.127,154.152,-69.141,175.270,21.009,153.381
C04335=1086.132,154.400,-69.162,175.272,21.011,153.381
C04336=1086.138,154.650,-69.183,175.275,21.013,153.381
C04337=1086.144,154.899,-69.204,175.277,21.015,153.381
C04338=1086.149,155.148,-69.225,175.280,21.016,153.381
C04339=1086.155,155.397,-69.246,175.281,21.017,153.381
C04340=1086.160,155.646,-69.267,175.284,21.019,153.381
C04341=1086.166,155.895,-69.288,175.286,21.021,153.381
C04342=1086.172,156.144,-69.309,175.289,21.023,153.381
C04343=1086.177,156.393,-69.330,175.291,21.024,153.381
C04344=1086.182,156.642,-69.351,175.294,21.026,153.381
C04345=1086.189,156.891,-69.373,175.295,21.027,153.381
C04346=1086.194,157.140,-69.393,175.298,21.029,153.381
C04347=1086.199,157.389,-69.414,175.300,21.031,153.381
C04348=1086.206,157.638,-69.436,175.303,21.032,153.380
C04349=1086.210,157.888,-69.457,175.305,21.034,153.380
C04350=1086.216,158.136,-69.478,175.308,21.035,153.380
C04351=1086.222,158.386,-69.499,175.309,21.037,153.380
C04352=1086.227,158.634,-69.521,175.312,21.038,153.380
C04353=1086.233,158.884,-69.542,175.314,21.040,153.380
C04354=1086.239,159.133,-69.563,175.317,21.042,153.380
C04355=1086.245,159.411,-69.588,175.319,21.044,153.380
C04356=1086.251,159.689,-69.611,175.322,21.045,153.380
C04357=1086.258,159.968,-69.634,175.325,21.047,153.380
C04358=1086.264,160.247,-69.658,175.328,21.049,153.380
C04359=1086.269,160.495,-69.680,175.330,21.051,153.380
C04360=1086.275,160.744,-69.701,175.332,21.052,153.380
C04361=1086.281,160.994,-69.722,175.334,21.053,153.380
C04362=1086.286,161.242,-69.743,175.337,21.055,153.380
C04363=1086.292,161.492,-69.765,175.339,21.057,153.380
C04364=1086.297,161.740,-69.787,175.342,21.059,153.380
C04365=1086.302,161.989,-69.807,175.344,21.061,153.380
C04366=1086.308,162.239,-69.829,175.347,21.062,153.380
C04367=1086.313,162.487,-69.851,175.348,21.063,153.380
C04368=1086.318,162.736,-69.873,175.351,21.065,153.380
C04369=1086.324,162.985,-69.894,175.353,21.067,153.380
C04370=1086.330,163.234,-69.915,175.356,21.069,153.380
C04371=1086.335,163.484,-69.937,175.358,21.071,153.380
C04372=1086.341,163.732,-69.958,175.361,21.072,153.379
C04373=1086.345,163.981,-69.980,175.363,21.074,153.380
C04374=1086.352,164.230,-70.002,175.366,21.075,153.379
C04375=1086.357,164.479,-70.023,175.367,21.077,153.379
C04376=1086.362,164.729,-70.044,175.370,21.079,153.379
C04377=1086.368,164.978,-70.066,175.372,21.080,153.379
C04378=1086.373,165.226,-70.088,175.375,21.082,153.379
C04379=1086.379,165.476,-70.109,175.377,21.083,153.379
C04380=1086.384,165.724,-70.131,175.380,21.085,153.379
C04381=1086.390,165.974,-70.153,175.382,21.087,153.379
C04382=1086.395,166.222,-70.175,175.385,21.089,153.379
C04383=1086.401,166.472,-70.196,175.387,21.090,153.379
C04384=1086.406,166.720,-70.218,175.389,21.091,153.379
C04385=1086.412,166.970,-70.240,175.391,21.093,153.379
C04386=1086.417,167.219,-70.262,175.394,21.095,153.379
C04387=1086.422,167.467,-70.283,175.396,21.097,153.379
C04388=1086.428,167.717,-70.305,175.399,21.098,153.379
C04389=1086.433,167.965,-70.326,175.401,21.100,153.379
C04390=1086.439,168.215,-70.349,175.404,21.101,153.379
C04391=1086.444,168.463,-70.370,175.406,21.103,153.379
C04392=1086.450,168.713,-70.392,175.409,21.105,153.379
C04393=1086.455,168.961,-70.413,175.411,21.107,153.379
C04394=1086.461,169.211,-70.436,175.414,21.108,153.379
C04395=1086.466,169.459,-70.457,175.415,21.109,153.379
C04396=1086.472,169.709,-70.479,175.418,21.111,153.378
C04397=1086.478,169.958,-70.501,175.420,21.113,153.379
C04398=1086.483,170.207,-70.523,175.423,21.114,153.378
C04399=1086.489,170.456,-70.544,175.425,21.116,153.378
C04400=1086.494,170.704,-70.567,175.428,21.117,153.378
C04401=1086.500,170.953,-70.588,175.430,21.119,153.378
C04402=1086.505,171.202,-70.610,175.433,21.121,153.378
C04403=1086.511,171.451,-70.632,175.435,21.122,153.378
C04404=1086.516,171.700,-70.654,175.438,21.124,153.378
C04405=1086.522,171.949,-70.675,175.440,21.125,153.378
C04406=1086.527,172.199,-70.698,175.443,21.127,153.378
C04407=1086.533,172.447,-70.720,175.445,21.128,153.378
C04408=1086.539,172.696,-70.742,175.447,21.130,153.378
C04409=1086.544,172.945,-70.764,175.450,21.132,153.378
C04410=1086.550,173.194,-70.785,175.452,21.133,153.378
C04411=1086.555,173.443,-70.808,175.455,21.135,153.378
C04412=1086.561,173.692,-70.830,175.457,21.136,153.378
C04413=1086.566,173.941,-70.852,175.460,21.138,153.378
C04414=1086.571,174.190,-70.874,175.462,21.140,153.377
C04415=1086.578,174.439,-70.896,175.465,21.141,153.377
C04416=1086.583,174.688,-70.918,175.467,21.143,153.377
C04417=1086.589,174.937,-70.940,175.470,21.144,153.377
C04418=1086.594,175.185,-70.963,175.472,21.146,153.377
C04419=1086.601,175.464,-70.987,175.475,21.148,153.377
C04420=1086.606,175.742,-71.012,175.477,21.149,153.377
C04421=1086.613,176.020,-71.037,175.481,21.151,153.377
C04422=1086.619,176.298,-71.061,175.483,21.153,153.377
C04423=1086.625,176.547,-71.083,175.486,21.154,153.377
C04424=1086.630,176.796,-71.106,175.488,21.156,153.377
C04425=1086.636,177.045,-71.127,175.491,21.158,153.377
C04426=1086.642,177.294,-71.150,175.493,21.159,153.377
C04427=1086.647,177.543,-71.172,175.496,21.161,153.377
C04428=1086.653,177.792,-71.194,175.498,21.162,153.376
C04429=1086.659,178.041,-71.217,175.501,21.164,153.376
C04430=1086.664,178.290,-71.239,175.503,21.166,153.376
C04431=1086.670,178.538,-71.261,175.506,21.167,153.376
C04432=1086.676,178.788,-71.283,175.509,21.168,153.376
C04433=1086.681,179.036,-71.306,175.511,21.170,153.376
C04434=1086.687,179.286,-71.328,175.514,21.172,153.376
C04435=1086.693,179.534,-71.350,175.516,21.173,153.376
C04436=1086.698,179.783,-71.372,175.519,21.175,153.376
C04437=1086.704,180.032,-71.395,175.521,21.176,153.376
C04438=1086.710,180.282,-71.417,175.524,21.178,153.376
C04439=1086.715,180.530,-71.440,175.526,21.179,153.376
C04440=1086.720,180.779,-71.462,175.528,21.180,153.376
C04441=1086.727,181.028,-71.484,175.531,21.182,153.375
C04442=1086.733,181.277,-71.507,175.533,21.183,153.375
C04443=1086.738,181.526,-71.529,175.536,21.185,153.375
C04444=1086.744,181.774,-71.551,175.538,21.186,153.375
C04445=1086.749,182.024,-71.574,175.541,21.188,153.375
C04446=1086.755,182.273,-71.597,175.543,21.190,153.375
C04447=1086.761,182.521,-71.619,175.546,21.191,153.375
C04448=1086.767,182.771,-71.641,175.549,21.192,153.375
C04449=1086.773,183.020,-71.664,175.551,21.194,153.375
C04450=1086.778,183.268,-71.687,175.554,21.195,153.375
C04451=1086.783,183.517,-71.709,175.556,21.197,153.374
C04452=1086.790,183.766,-71.731,175.559,21.199,153.375
C04453=1086.795,184.015,-71.754,175.561,21.200,153.374
C04454=1086.801,184.264,-71.776,175.564,21.201,153.374
C04455=1086.807,184.513,-71.799,175.567,21.203,153.374
C04456=1086.813,184.762,-71.822,175.569,21.204,153.374
C04457=1086.819,185.011,-71.844,175.572,21.206,153.374
C04458=1086.824,185.259,-71.866,175.575,21.208,153.374
C04459=1086.829,185.508,-71.889,175.578,21.209,153.374
C04460=1086.835,185.757,-71.912,175.580,21.211,153.374
C04461=1086.841,186.006,-71.935,175.583,21.213,153.374
C04462=1086.845,186.255,-71.958,175.585,21.214,153.374
C04463=1086.851,186.504,-71.981,175.588,21.216,153.374
C04464=1086.856,186.753,-72.004,175.590,21.217,153.373
C04465=1086.862,187.002,-72.027,175.593,21.219,153.373
C04466=1086.868,187.251,-72.050,175.595,21.221,153.373
C04467=1086.873,187.500,-72.071,175.598,21.222,153.373
C04468=1086.878,187.749,-72.094,175.600,21.224,153.373
C04469=1086.884,187.997,-72.117,175.603,21.225,153.373
C04470=1086.889,188.247,-72.141,175.606,21.227,153.373
C04471=1086.895,188.496,-72.164,175.608,21.229,153.373
C04472=1086.900,188.744,-72.186,175.611,21.230,153.373
C04473=1086.906,188.993,-72.209,175.613,21.231,153.373
C04474=1086.911,189.242,-72.232,175.616,21.233,153.373
C04475=1086.917,189.490,-72.255,175.618,21.235,153.373
C04476=1086.922,189.740,-72.278,175.621,21.236,153.373
C04477=1086.928,189.989,-72.301,175.623,21.238,153.373
C04478=1086.933,190.237,-72.324,175.626,21.239,153.373
C04479=1086.938,190.486,-72.347,175.628,21.241,153.372
C04480=1086.944,190.735,-72.369,175.631,21.242,153.372
C04481=1086.950,190.984,-72.392,175.633,21.244,153.372
C04482=1086.955,191.233,-72.416,175.637,21.246,153.372
C04483=1086.962,191.511,-72.441,175.640,21.247,153.372
C04484=1086.967,191.789,-72.468,175.642,21.249,153.372
C04485=1086.973,192.066,-72.493,175.645,21.251,153.372
C04486=1086.980,192.344,-72.518,175.648,21.253,153.372
C04487=1086.985,192.592,-72.543,175.651,21.254,153.372
C04488=1086.991,192.841,-72.565,175.653,21.256,153.372
C04489=1086.997,193.090,-72.588,175.656,21.257,153.372
C04490=1087.002,193.339,-72.611,175.659,21.259,153.371
C04491=1087.007,193.588,-72.635,175.662,21.261,153.371
C04492=1087.013,193.837,-72.658,175.664,21.263,153.371
C04493=1087.019,194.086,-72.681,175.667,21.264,153.371
C04494=1087.025,194.335,-72.704,175.669,21.265,153.371
C04495=1087.030,194.584,-72.727,175.672,21.267,153.371
C04496=1087.036,194.833,-72.751,175.674,21.269,153.371
C04497=1087.041,195.081,-72.774,175.677,21.270,153.371
C04498=1087.047,195.330,-72.797,175.680,21.271,153.371
C04499=1087.052,195.580,-72.820,175.682,21.273,153.371
C04500=1087.058,195.828,-72.843,175.685,21.274,153.371
C04501=1087.064,196.077,-72.867,175.687,21.276,153.371
C04502=1087.070,196.326,-72.890,175.691,21.278,153.370
C04503=1087.075,196.575,-72.913,175.693,21.279,153.370
C04504=1087.080,196.824,-72.936,175.696,21.281,153.370
C04505=1087.086,197.072,-72.960,175.698,21.282,153.370
C04506=1087.091,197.321,-72.984,175.701,21.284,153.370
C04507=1087.097,197.570,-73.007,175.703,21.286,153.370
C04508=1087.103,197.819,-73.029,175.706,21.287,153.370
C04509=1087.109,198.067,-73.053,175.709,21.288,153.370
C04510=1087.114,198.316,-73.077,175.711,21.290,153.370
C04511=1087.120,198.565,-73.100,175.715,21.292,153.370
C04512=1087.126,198.814,-73.123,175.717,21.293,153.369
C04513=1087.131,199.063,-73.147,175.720,21.295,153.369
C04514=1087.137,199.311,-73.171,175.722,21.296,153.369
C04515=1087.143,199.561,-73.194,175.725,21.298,153.369
C04516=1087.148,199.810,-73.217,175.728,21.299,153.369
C04517=1087.154,200.058,-73.241,175.730,21.301,153.369
C04518=1087.160,200.307,-73.264,175.733,21.302,153.369
C04519=1087.165,200.556,-73.288,175.736,21.304,153.369
C04520=1087.171,200.805,-73.311,175.739,21.306,153.369
C04521=1087.176,201.054,-73.335,175.741,21.307,153.369
C04522=1087.182,201.302,-73.358,175.744,21.309,153.369
C04523=1087.188,201.552,-73.382,175.747,21.310,153.368
C04524=1087.193,201.800,-73.406,175.749,21.311,153.368
C04525=1087.199,202.049,-73.429,175.752,21.313,153.368
C04526=1087.205,202.297,-73.453,175.755,21.315,153.368
C04527=1087.210,202.547,-73.476,175.758,21.316,153.368
C04528=1087.216,202.795,-73.500,175.760,21.317,153.368
C04529=1087.221,203.044,-73.523,175.763,21.319,153.368
C04530=1087.228,203.293,-73.547,175.765,21.321,153.368
C04531=1087.233,203.542,-73.572,175.768,21.322,153.368
C04532=1087.238,203.791,-73.595,175.771,21.324,153.368
C04533=1087.244,204.039,-73.619,175.774,21.325,153.367
C04534=1087.249,204.288,-73.642,175.777,21.327,153.367
C04535=1087.255,204.537,-73.666,175.779,21.329,153.367
C04536=1087.260,204.786,-73.690,175.782,21.330,153.367
C04537=1087.266,205.034,-73.714,175.784,21.332,153.367
C04538=1087.272,205.283,-73.738,175.787,21.333,153.367
C04539=1087.277,205.533,-73.761,175.790,21.335,153.367
C04540=1087.282,205.781,-73.786,175.793,21.337,153.367
C04541=1087.289,206.029,-73.809,175.796,21.338,153.367
C04542=1087.294,206.279,-73.833,175.798,21.339,153.367
C04543=1087.300,206.527,-73.856,175.801,21.341,153.367
C04544=1087.305,206.776,-73.881,175.803,21.343,153.367
C04545=1087.311,207.025,-73.905,175.807,21.345,153.366
C04546=1087.316,207.274,-73.928,175.809,21.346,153.366
C04547=1087.339,208.299,-74.028,175.886,21.385,153.363
C04548=1087.348,208.684,-74.065,175.889,21.389,153.363
C04549=1087.357,209.069,-74.103,175.894,21.393,153.363
C04550=1087.365,209.454,-74.141,175.898,21.397,153.363
C04551=1087.375,209.840,-74.179,175.902,21.401,153.363
C04552=1087.380,210.088,-74.203,175.905,21.403,153.364
C04553=1087.385,210.337,-74.227,175.907,21.405,153.364
C04554=1087.391,210.586,-74.252,175.909,21.408,153.364
C04555=1087.397,210.835,-74.276,175.912,21.411,153.364
C04556=1087.402,211.084,-74.301,175.914,21.413,153.364
C04557=1087.408,211.332,-74.326,175.918,21.415,153.364
C04558=1087.413,211.581,-74.350,175.920,21.418,153.364
C04559=1087.419,211.830,-74.375,175.923,21.421,153.364
C04560=1087.425,212.078,-74.399,175.925,21.423,153.365
C04561=1087.430,212.328,-74.423,175.927,21.425,153.365
C04562=1087.436,212.576,-74.448,175.931,21.428,153.365
C04563=1087.441,212.824,-74.473,175.933,21.430,153.365
C04564=1087.447,213.074,-74.497,175.936,21.433,153.365
C04565=1087.453,213.322,-74.522,175.938,21.435,153.365
C04566=1087.459,213.571,-74.547,175.941,21.438,153.365
C04567=1087.464,213.819,-74.571,175.944,21.440,153.365
C04568=1087.470,214.069,-74.596,175.947,21.443,153.366
C04569=1087.476,214.317,-74.621,175.949,21.445,153.366
C04570=1087.481,214.566,-74.646,175.952,21.448,153.366
C04571=1087.486,214.814,-74.671,175.954,21.451,153.366
C04572=1087.492,215.063,-74.695,175.957,21.452,153.366
C04573=1087.498,215.312,-74.720,175.960,21.455,153.366
C04574=1087.503,215.560,-74.745,175.962,21.458,153.366
C04575=1087.509,215.809,-74.769,175.965,21.461,153.366
C04576=1087.514,216.058,-74.794,175.967,21.463,153.367
C04577=1087.520,216.307,-74.820,175.970,21.465,153.367
C04578=1087.525,216.555,-74.844,175.973,21.468,153.367
C04579=1087.531,216.804,-74.869,175.976,21.471,153.367
C04580=1087.537,217.053,-74.893,175.978,21.473,153.367
C04581=1087.543,217.301,-74.919,175.981,21.476,153.367
C04582=1087.547,217.550,-74.944,175.983,21.478,153.367
C04583=1087.554,217.799,-74.969,175.986,21.481,153.367
C04584=1087.559,218.048,-74.993,175.989,21.483,153.368
C04585=1087.565,218.296,-75.019,175.992,21.486,153.368
C04586=1087.571,218.546,-75.043,175.994,21.488,153.368
C04587=1087.576,218.794,-75.069,175.997,21.491,153.368
C04588=1087.582,219.043,-75.093,175.999,21.493,153.368
C04589=1087.587,219.291,-75.118,176.002,21.496,153.368
C04590=1087.594,219.540,-75.144,176.005,21.498,153.368
C04591=1087.599,219.788,-75.168,176.007,21.500,153.368
C04592=1087.604,220.037,-75.194,176.010,21.503,153.369
C04593=1087.611,220.286,-75.219,176.012,21.505,153.369
C04594=1087.616,220.535,-75.243,176.015,21.508,153.369
C04595=1087.622,220.783,-75.269,176.018,21.510,153.369
C04596=1087.627,221.032,-75.294,176.021,21.513,153.369
C04597=1087.633,221.281,-75.319,176.023,21.515,153.369
C04598=1087.639,221.529,-75.344,176.026,21.518,153.369
C04599=1087.644,221.778,-75.370,176.029,21.520,153.369
C04600=1087.653,222.167,-75.408,176.033,21.524,153.370
C04601=1087.662,222.557,-75.448,176.037,21.528,153.370
C04602=1087.670,222.945,-75.488,176.042,21.532,153.370
C04603=1087.679,223.334,-75.528,176.045,21.536,153.370
C04604=1087.684,223.583,-75.553,176.048,21.539,153.370
C04605=1087.690,223.831,-75.578,176.051,21.541,153.371
C04606=1087.696,224.081,-75.603,176.054,21.544,153.371
C04607=1087.701,224.329,-75.629,176.056,21.546,153.371
C04608=1087.707,224.578,-75.654,176.059,21.549,153.371
C04609=1087.713,224.826,-75.680,176.061,21.551,153.371
C04610=1087.719,225.074,-75.705,176.064,21.554,153.371
C04611=1087.724,225.323,-75.731,176.067,21.557,153.371
C04612=1087.730,225.572,-75.756,176.070,21.559,153.371
C04613=1087.735,225.821,-75.781,176.073,21.562,153.371
C04614=1087.741,226.070,-75.806,176.075,21.564,153.372
C04615=1087.746,226.319,-75.832,176.078,21.567,153.372
C04616=1087.752,226.567,-75.857,176.080,21.569,153.372
C04617=1087.758,226.816,-75.883,176.084,21.572,153.372
C04618=1087.764,227.064,-75.908,176.086,21.574,153.372
C04619=1087.769,227.313,-75.934,176.089,21.577,153.372
C04620=1087.775,227.561,-75.959,176.091,21.579,153.372
C04621=1087.780,227.810,-75.985,176.094,21.582,153.373
C04622=1087.786,228.059,-76.011,176.097,21.584,153.373
C04623=1087.791,228.307,-76.036,176.100,21.587,153.373
C04624=1087.797,228.556,-76.062,176.102,21.589,153.373
C04625=1087.803,228.805,-76.088,176.105,21.592,153.373
C04626=1087.808,229.054,-76.113,176.108,21.595,153.373
C04627=1087.815,229.302,-76.139,176.111,21.597,153.373
C04628=1087.820,229.550,-76.165,176.114,21.600,153.373
C04629=1087.826,229.799,-76.190,176.116,21.602,153.374
C04630=1087.832,230.048,-76.216,176.119,21.605,153.374
C04631=1087.837,230.297,-76.242,176.121,21.607,153.374
C04632=1087.843,230.545,-76.267,176.124,21.610,153.374
C04633=1087.848,230.794,-76.293,176.127,21.612,153.374
C04634=1087.854,231.043,-76.319,176.130,21.615,153.374
C04635=1087.860,231.291,-76.345,176.133,21.618,153.374
C04636=1087.866,231.540,-76.371,176.135,21.620,153.374
C04637=1087.870,231.788,-76.397,176.138,21.623,153.375
C04638=1087.876,232.037,-76.423,176.141,21.625,153.375
C04639=1087.882,232.285,-76.449,176.144,21.628,153.375
C04640=1087.888,232.534,-76.475,176.146,21.630,153.375
C04641=1087.893,232.783,-76.501,176.149,21.633,153.375
C04642=1087.898,233.031,-76.526,176.152,21.636,153.375
C04643=1087.905,233.279,-76.552,176.154,21.638,153.375
C04644=1087.910,233.528,-76.578,176.157,21.641,153.376
C04645=1087.916,233.777,-76.604,176.160,21.643,153.376
C04646=1087.921,234.026,-76.631,176.163,21.646,153.376
C04647=1087.927,234.275,-76.657,176.165,21.648,153.376
C04648=1087.932,234.523,-76.682,176.168,21.651,153.376
C04649=1087.938,234.771,-76.708,176.171,21.654,153.376
C04650=1087.944,235.020,-76.734,176.173,21.656,153.376
C04651=1087.949,235.269,-76.760,176.176,21.659,153.376
C04652=1087.958,235.649,-76.801,176.180,21.663,153.377
C04653=1087.966,236.030,-76.840,176.185,21.667,153.377
C04654=1087.975,236.410,-76.881,176.189,21.670,153.377
C04655=1087.984,236.790,-76.920,176.193,21.675,153.377
C04656=1087.989,237.039,-76.946,176.196,21.677,153.377
C04657=1087.995,237.287,-76.973,176.199,21.680,153.378
C04658=1088.000,237.536,-76.999,176.202,21.683,153.378
C04659=1088.006,237.784,-77.026,176.204,21.685,153.378
C04660=1088.012,238.033,-77.051,176.207,21.688,153.378
C04661=1088.017,238.282,-77.078,176.210,21.690,153.378
C04662=1088.023,238.531,-77.104,176.213,21.693,153.378
C04663=1088.029,238.779,-77.131,176.216,21.695,153.378
C04664=1088.034,239.028,-77.157,176.218,21.698,153.379
C04665=1088.040,239.276,-77.183,176.221,21.701,153.379
C04666=1088.046,239.525,-77.210,176.223,21.703,153.379
C04667=1088.051,239.774,-77.236,176.226,21.706,153.379
C04668=1088.057,240.022,-77.263,176.230,21.708,153.379
C04669=1088.063,240.271,-77.289,176.232,21.711,153.379
C04670=1088.068,240.520,-77.315,176.235,21.713,153.379
C04671=1088.074,240.768,-77.342,176.238,21.716,153.379
C04672=1088.080,241.016,-77.368,176.240,21.719,153.380
C04673=1088.085,241.265,-77.394,176.243,21.721,153.380
C04674=1088.091,241.514,-77.421,176.246,21.724,153.380
C04675=1088.097,241.762,-77.448,176.249,21.727,153.380
C04676=1088.102,242.011,-77.474,176.252,21.729,153.380
C04677=1088.108,242.259,-77.500,176.254,21.731,153.380
C04678=1088.114,242.508,-77.527,176.257,21.734,153.380
C04679=1088.120,242.756,-77.553,176.260,21.737,153.381
C04680=1088.125,243.004,-77.580,176.263,21.739,153.381
C04681=1088.131,243.253,-77.606,176.266,21.742,153.381
C04682=1088.137,243.502,-77.633,176.269,21.745,153.381
C04683=1088.142,243.750,-77.660,176.271,21.747,153.381
C04684=1088.147,243.999,-77.687,176.274,21.750,153.381
C04685=1088.153,244.247,-77.713,176.276,21.753,153.382
C04686=1088.159,244.495,-77.740,176.279,21.755,153.382
C04687=1088.164,244.744,-77.767,176.282,21.758,153.382
C04688=1088.169,244.993,-77.793,176.285,21.761,153.382
C04689=1088.175,245.241,-77.820,176.288,21.763,153.382
C04690=1088.181,245.490,-77.846,176.291,21.766,153.382
C04691=1088.187,245.738,-77.873,176.293,21.768,153.382
C04692=1088.192,245.987,-77.900,176.296,21.771,153.382
C04693=1088.198,246.235,-77.927,176.299,21.774,153.383
C04694=1088.203,246.484,-77.954,176.302,21.776,153.383
C04695=1088.209,246.732,-77.980,176.305,21.779,153.383
C04696=1088.215,246.981,-78.008,176.308,21.782,153.383
C04697=1088.221,247.230,-78.034,176.310,21.784,153.383
C04698=1088.226,247.478,-78.061,176.313,21.787,153.383
C04699=1088.231,247.727,-78.088,176.316,21.790,153.384
C04700=1088.237,247.975,-78.115,176.318,21.792,153.384
C04701=1088.242,248.224,-78.142,176.322,21.795,153.384
C04702=1088.248,248.472,-78.169,176.325,21.798,153.384
C04703=1088.253,248.720,-78.197,176.327,21.800,153.384
C04704=1088.262,249.094,-78.237,176.332,21.805,153.384
C04705=1088.270,249.468,-78.278,176.335,21.808,153.385
C04706=1088.278,249.841,-78.318,176.340,21.813,153.385
C04707=1088.286,250.214,-78.360,176.344,21.817,153.385
C04708=1088.292,250.463,-78.386,176.347,21.820,153.385
C04709=1088.298,250.712,-78.414,176.350,21.823,153.386
C04710=1088.304,250.960,-78.440,176.353,21.825,153.386
C04711=1088.309,251.209,-78.467,176.355,21.828,153.386
C04712=1088.315,251.457,-78.495,176.358,21.831,153.386
C04713=1088.320,251.705,-78.522,176.361,21.833,153.386
C04714=1088.326,251.954,-78.549,176.363,21.836,153.386
C04715=1088.331,252.202,-78.577,176.367,21.839,153.387
C04716=1088.337,252.451,-78.604,176.370,21.841,153.387
C04717=1088.342,252.700,-78.631,176.373,21.844,153.387
C04718=1088.348,252.947,-78.658,176.375,21.847,153.387
C04719=1088.353,253.196,-78.686,176.378,21.849,153.387
C04720=1088.359,253.444,-78.712,176.381,21.852,153.387
C04721=1088.365,253.693,-78.741,176.383,21.855,153.387
C04722=1088.371,253.942,-78.767,176.386,21.857,153.388
C04723=1088.376,254.190,-78.795,176.390,21.860,153.388
C04724=1088.382,254.438,-78.822,176.393,21.863,153.388
C04725=1088.388,254.687,-78.850,176.395,21.865,153.388
C04726=1088.393,254.935,-78.878,176.398,21.868,153.388
C04727=1088.399,255.184,-78.904,176.401,21.871,153.388
C04728=1088.404,255.432,-78.932,176.403,21.873,153.389
C04729=1088.411,255.681,-78.959,176.406,21.876,153.389
C04730=1088.416,255.929,-78.987,176.410,21.879,153.389
C04731=1088.422,256.177,-79.014,176.413,21.882,153.389
C04732=1088.428,256.426,-79.042,176.415,21.884,153.389
C04733=1088.433,256.675,-79.069,176.418,21.887,153.389
C04734=1088.439,256.922,-79.097,176.421,21.890,153.390
C04735=1088.444,257.172,-79.124,176.423,21.892,153.390
C04736=1088.450,257.419,-79.152,176.426,21.895,153.390
C04737=1088.455,257.668,-79.179,176.429,21.898,153.390
C04738=1088.461,257.917,-79.207,176.433,21.901,153.390
C04739=1088.467,258.165,-79.235,176.435,21.903,153.390
C04740=1088.473,258.413,-79.262,176.438,21.906,153.390
C04741=1088.478,258.662,-79.290,176.441,21.909,153.391
C04742=1088.485,258.910,-79.318,176.444,21.912,153.391
C04743=1088.490,259.158,-79.345,176.446,21.914,153.391
C04744=1088.496,259.407,-79.373,176.449,21.917,153.391
C04745=1088.502,259.655,-79.400,176.453,21.920,153.391
C04746=1088.507,259.904,-79.428,176.456,21.922,153.391
C04747=1088.513,260.152,-79.456,176.458,21.925,153.392
C04748=1088.519,260.400,-79.483,176.461,21.927,153.392
C04749=1088.525,260.649,-79.512,176.464,21.930,153.392
C04750=1088.530,260.898,-79.539,176.467,21.933,153.392
C04751=1088.536,261.146,-79.567,176.469,21.935,153.392
C04752=1088.542,261.394,-79.595,176.473,21.938,153.392
C04753=1088.547,261.642,-79.623,176.476,21.941,153.393
C04754=1088.553,261.891,-79.650,176.479,21.944,153.393
C04755=1088.559,262.139,-79.678,176.481,21.946,153.393
C04756=1088.567,262.510,-79.720,176.486,21.951,153.393
C04757=1088.576,262.881,-79.761,176.490,21.955,153.393
C04758=1088.585,263.251,-79.803,176.494,21.959,153.394
C04759=1088.593,263.622,-79.845,176.499,21.963,153.394
C04760=1088.599,263.870,-79.873,176.502,21.966,153.394
C04761=1088.605,264.118,-79.900,176.504,21.968,153.394
C04762=1088.611,264.367,-79.929,176.507,21.971,153.394
C04763=1088.616,264.615,-79.957,176.510,21.974,153.395
C04764=1088.622,264.864,-79.984,176.513,21.977,153.395
C04765=1088.627,265.112,-80.012,176.516,21.980,153.395
C04766=1088.634,265.360,-80.041,176.519,21.982,153.395
C04767=1088.639,265.608,-80.069,176.522,21.985,153.395
C04768=1088.645,265.857,-80.098,176.525,21.988,153.395
C04769=1088.650,266.105,-80.126,176.528,21.991,153.396
C04770=1088.656,266.354,-80.154,176.530,21.993,153.396
C04771=1088.662,266.602,-80.182,176.533,21.996,153.396
C04772=1088.668,266.851,-80.210,176.536,21.999,153.396
C04773=1088.673,267.099,-80.238,176.539,22.002,153.396
C04774=1088.679,267.348,-80.266,176.542,22.005,153.396
C04775=1088.684,267.596,-80.294,176.544,22.007,153.397
C04776=1088.690,267.844,-80.323,176.547,22.010,153.397
C04777=1088.696,268.092,-80.351,176.551,22.013,153.397
C04778=1088.702,268.341,-80.380,176.554,22.016,153.397
C04779=1088.707,268.589,-80.408,176.557,22.019,153.397
C04780=1088.713,268.837,-80.436,176.560,22.021,153.398
C04781=1088.718,269.085,-80.464,176.562,22.024,153.398
C04782=1088.724,269.334,-80.494,176.565,22.027,153.398
C04783=1088.729,269.582,-80.522,176.568,22.030,153.398
C04784=1088.735,269.831,-80.550,176.571,22.033,153.398
C04785=1088.741,270.079,-80.578,176.574,22.035,153.398
C04786=1088.747,270.327,-80.607,176.576,22.038,153.399
C04787=1088.753,270.576,-80.635,176.580,22.041,153.399
C04788=1088.758,270.824,-80.663,176.583,22.044,153.399
C04789=1088.764,271.072,-80.693,176.586,22.047,153.399
C04790=1088.769,271.320,-80.721,176.589,22.050,153.400
C04791=1088.775,271.569,-80.749,176.592,22.053,153.400
C04792=1088.781,271.817,-80.778,176.594,22.055,153.400
C04793=1088.786,272.065,-80.806,176.597,22.058,153.400
C04794=1088.793,272.313,-80.835,176.600,22.061,153.400
C04795=1088.797,272.562,-80.864,176.603,22.064,153.400
C04796=1088.803,272.810,-80.892,176.606,22.067,153.401
C04797=1088.809,273.059,-80.921,176.609,22.069,153.401
C04798=1088.815,273.307,-80.949,176.611,22.073,153.401
C04799=1088.820,273.555,-80.979,176.615,22.075,153.401
C04800=1088.826,273.804,-81.007,176.618,22.078,153.401
C04801=1088.832,274.051,-81.036,176.621,22.081,153.402
C04802=1088.838,274.300,-81.064,176.624,22.084,153.402
C04803=1088.843,274.548,-81.094,176.627,22.087,153.402
C04804=1088.849,274.796,-81.122,176.629,22.089,153.402
C04805=1088.855,275.045,-81.151,176.632,22.093,153.402
C04806=1088.860,275.293,-81.179,176.635,22.095,153.403
C04807=1088.866,275.541,-81.208,176.638,22.098,153.403
C04808=1088.874,275.915,-81.252,176.643,22.103,153.403
C04809=1088.883,276.288,-81.295,176.647,22.107,153.403
C04810=1088.891,276.662,-81.339,176.651,22.111,153.404
C04811=1088.900,277.035,-81.383,176.656,22.116,153.404
C04812=1088.906,277.283,-81.411,176.659,22.119,153.404
C04813=1088.911,277.532,-81.440,176.662,22.122,153.404
C04814=1088.917,277.780,-81.469,176.665,22.125,153.405
C04815=1088.923,278.029,-81.498,176.668,22.128,153.405
C04816=1088.928,278.276,-81.527,176.671,22.131,153.405
C04817=1088.934,278.525,-81.557,176.673,22.133,153.405
C04818=1088.940,278.773,-81.586,176.676,22.136,153.406
C04819=1088.945,279.021,-81.614,176.679,22.139,153.406
C04820=1088.951,279.269,-81.643,176.682,22.142,153.406
C04821=1088.956,279.518,-81.673,176.685,22.145,153.406
C04822=1088.963,279.766,-81.702,176.688,22.148,153.406
C04823=1088.968,280.014,-81.731,176.691,22.151,153.407
C04824=1088.974,280.262,-81.760,176.694,22.154,153.407
C04825=1088.980,280.510,-81.788,176.696,22.157,153.407
C04826=1088.985,280.759,-81.818,176.700,22.160,153.407
C04827=1088.991,281.007,-81.848,176.703,22.162,153.407
C04828=1088.996,281.255,-81.876,176.706,22.166,153.408
C04829=1089.002,281.503,-81.906,176.709,22.168,153.408
C04830=1089.008,281.751,-81.935,176.712,22.172,153.408
C04831=1089.014,282.000,-81.965,176.715,22.175,153.408
C04832=1089.019,282.247,-81.994,176.718,22.178,153.409
C04833=1089.025,282.496,-82.023,176.721,22.181,153.409
C04834=1089.030,282.744,-82.053,176.724,22.184,153.409
C04835=1089.036,282.993,-82.082,176.726,22.186,153.409
C04836=1089.042,283.241,-82.111,176.729,22.190,153.410
C04837=1089.047,283.488,-82.141,176.732,22.192,153.410
C04838=1089.053,283.737,-82.170,176.735,22.196,153.410
C04839=1089.059,283.985,-82.199,176.738,22.198,153.410
C04840=1089.064,284.233,-82.229,176.741,22.202,153.410
C04841=1089.070,284.482,-82.259,176.744,22.204,153.411
C04842=1089.076,284.730,-82.288,176.747,22.208,153.411
C04843=1089.081,284.977,-82.318,176.750,22.211,153.411
C04844=1089.087,285.226,-82.347,176.753,22.214,153.411
C04845=1089.092,285.474,-82.377,176.756,22.217,153.412
C04846=1089.099,285.722,-82.406,176.759,22.220,153.412
C04847=1089.104,285.971,-82.436,176.761,22.223,153.412
C04848=1089.110,286.219,-82.465,176.764,22.226,153.412
C04849=1089.115,286.467,-82.496,176.767,22.229,153.413
C04850=1089.122,286.715,-82.525,176.770,22.232,153.413
C04851=1089.127,286.963,-82.554,176.773,22.235,153.413
C04852=1089.132,287.211,-82.583,176.777,22.238,153.413
C04853=1089.138,287.459,-82.614,176.779,22.241,153.414
C04854=1089.144,287.707,-82.643,176.783,22.244,153.414
C04855=1089.150,287.956,-82.672,176.785,22.247,153.414
C04856=1089.155,288.203,-82.703,176.789,22.250,153.414
C04857=1089.161,288.452,-82.732,176.792,22.253,153.414
C04858=1089.167,288.700,-82.762,176.795,22.256,153.415
C04859=1089.173,288.948,-82.792,176.798,22.259,153.415
C04860=1089.182,289.331,-82.838,176.802,22.264,153.415
C04861=1089.190,289.715,-82.884,176.807,22.268,153.416
C04862=1089.199,290.097,-82.930,176.811,22.273,153.416
C04863=1089.208,290.480,-82.976,176.816,22.278,153.416
C04864=1089.214,290.728,-83.006,176.819,22.281,153.417
C04865=1089.220,290.976,-83.036,176.822,22.284,153.417
C04866=1089.225,291.224,-83.066,176.825,22.287,153.417
C04867=1089.231,291.472,-83.096,176.828,22.290,153.417
C04868=1089.237,291.720,-83.126,176.831,22.293,153.418
C04869=1089.242,291.969,-83.156,176.834,22.296,153.418
C04870=1089.248,292.216,-83.186,176.837,22.300,153.418
C04871=1089.254,292.465,-83.216,176.840,22.303,153.419
C04872=1089.259,292.713,-83.246,176.843,22.306,153.419
C04873=1089.265,292.961,-83.276,176.846,22.309,153.419
C04874=1089.271,293.209,-83.306,176.849,22.312,153.419
C04875=1089.277,293.457,-83.336,176.852,22.315,153.419
C04876=1089.282,293.705,-83.366,176.855,22.318,153.420
C04877=1089.288,293.953,-83.396,176.858,22.322,153.420
C04878=1089.294,294.201,-83.427,176.860,22.325,153.420
C04879=1089.298,294.450,-83.457,176.864,22.328,153.421
C04880=1089.304,294.697,-83.487,176.867,22.331,153.421
C04881=1089.310,294.945,-83.518,176.870,22.334,153.421
C04882=1089.316,295.193,-83.548,176.872,22.337,153.421
C04883=1089.322,295.442,-83.578,176.876,22.340,153.422
C04884=1089.328,295.690,-83.608,176.879,22.343,153.422
C04885=1089.334,295.938,-83.639,176.881,22.347,153.422
C04886=1089.340,296.186,-83.669,176.884,22.350,153.422
C04887=1089.345,296.434,-83.699,176.887,22.353,153.423
C04888=1089.351,296.682,-83.729,176.890,22.356,153.423
C04889=1089.356,296.930,-83.760,176.893,22.359,153.423
C04890=1089.362,297.178,-83.790,176.896,22.363,153.424
C04891=1089.368,297.426,-83.821,176.899,22.366,153.424
C04892=1089.373,297.674,-83.851,176.902,22.369,153.424
C04893=1089.380,297.922,-83.882,176.905,22.372,153.424
C04894=1089.385,298.171,-83.912,176.908,22.375,153.425
C04895=1089.390,298.419,-83.942,176.911,22.378,153.425
C04896=1089.396,298.666,-83.973,176.914,22.382,153.425
C04897=1089.401,298.915,-84.004,176.917,22.385,153.426
C04898=1089.407,299.162,-84.034,176.920,22.388,153.426
C04899=1089.412,299.411,-84.065,176.923,22.391,153.426
C04900=1089.418,299.658,-84.095,176.926,22.395,153.427
C04901=1089.424,299.906,-84.126,176.929,22.398,153.427
C04902=1089.429,300.154,-84.156,176.932,22.402,153.427
C04903=1089.435,300.403,-84.187,176.935,22.405,153.427
C04904=1089.440,300.651,-84.218,176.938,22.408,153.428
C04905=1089.447,300.898,-84.249,176.941,22.412,153.428
C04906=1089.452,301.146,-84.280,176.944,22.415,153.428
C04907=1089.457,301.394,-84.311,176.947,22.418,153.429
C04908=1089.463,301.642,-84.341,176.950,22.422,153.429
C04909=1089.468,301.890,-84.372,176.953,22.425,153.429
C04910=1089.475,302.139,-84.403,176.956,22.428,153.430
C04911=1089.480,302.387,-84.433,176.959,22.431,153.430
C04912=1089.489,302.784,-84.483,176.964,22.437,153.430
C04913=1089.498,303.181,-84.532,176.969,22.442,153.431
C04914=1089.507,303.577,-84.581,176.973,22.447,153.431
C04915=1089.516,303.974,-84.631,176.978,22.453,153.432
C04916=1089.522,304.222,-84.662,176.981,22.456,153.432
C04917=1089.528,304.470,-84.693,176.984,22.459,153.432
C04918=1089.533,304.719,-84.724,176.987,22.463,153.433
C04919=1089.539,304.966,-84.755,176.990,22.466,153.433
C04920=1089.544,305.214,-84.786,176.993,22.469,153.433
C04921=1089.550,305.462,-84.817,176.997,22.473,153.434
C04922=1089.556,305.710,-84.848,177.000,22.476,153.434
C04923=1089.562,305.958,-84.879,177.003,22.480,153.434
C04924=1089.567,306.207,-84.910,177.006,22.483,153.435
C04925=1089.573,306.454,-84.941,177.009,22.486,153.435
C04926=1089.578,306.702,-84.972,177.011,22.489,153.435
C04927=1089.585,306.950,-85.004,177.014,22.493,153.436
C04928=1089.590,307.198,-85.035,177.017,22.496,153.436
C04929=1089.596,307.445,-85.066,177.020,22.500,153.436
C04930=1089.601,307.693,-85.097,177.023,22.503,153.437
C04931=1089.607,307.942,-85.129,177.027,22.507,153.437
C04932=1089.613,308.189,-85.159,177.030,22.510,153.437
C04933=1089.619,308.438,-85.191,177.033,22.513,153.438
C04934=1089.625,308.685,-85.221,177.036,22.516,153.438
C04935=1089.630,308.933,-85.253,177.039,22.520,153.438
C04936=1089.636,309.182,-85.284,177.042,22.523,153.439
C04937=1089.642,309.429,-85.315,177.045,22.527,153.439
C04938=1089.648,309.678,-85.347,177.047,22.530,153.439
C04939=1089.653,309.925,-85.378,177.051,22.534,153.439
C04940=1089.659,310.172,-85.409,177.054,22.537,153.440
C04941=1089.665,310.421,-85.441,177.057,22.540,153.440
C04942=1089.671,310.669,-85.472,177.060,22.544,153.441
C04943=1089.677,310.917,-85.504,177.063,22.547,153.441
C04944=1089.682,311.165,-85.535,177.066,22.551,153.441
C04945=1089.688,311.413,-85.567,177.069,22.554,153.442
C04946=1089.694,311.660,-85.598,177.072,22.557,153.442
C04947=1089.700,311.908,-85.630,177.076,22.561,153.442
C04948=1089.706,312.157,-85.661,177.079,22.564,153.442
C04949=1089.712,312.405,-85.692,177.081,22.568,153.443
C04950=1089.718,312.652,-85.724,177.084,22.571,153.443
C04951=1089.724,312.900,-85.756,177.087,22.574,153.444
C04952=1089.729,313.148,-85.786,177.090,22.578,153.444
C04953=1089.735,313.396,-85.818,177.093,22.581,153.444
C04954=1089.741,313.644,-85.850,177.097,22.585,153.445
C04955=1089.747,313.892,-85.882,177.100,22.588,153.445
C04956=1089.753,314.139,-85.913,177.103,22.592,153.445
C04957=1089.759,314.387,-85.945,177.106,22.595,153.446
C04958=1089.765,314.636,-85.977,177.108,22.598,153.446
C04959=1089.770,314.883,-86.009,177.111,22.602,153.446
C04960=1089.777,315.132,-86.039,177.114,22.605,153.447
C04961=1089.781,315.379,-86.072,177.118,22.609,153.447
C04962=1089.787,315.628,-86.104,177.121,22.613,153.447
C04963=1089.793,315.875,-86.135,177.124,22.616,153.448
C04964=1089.802,316.275,-86.187,177.129,22.622,153.448
C04965=1089.811,316.675,-86.239,177.133,22.628,153.449
C04966=1089.821,317.074,-86.290,177.138,22.634,153.450
C04967=1089.829,317.474,-86.341,177.143,22.640,153.450
C04968=1089.835,317.722,-86.373,177.146,22.643,153.451
C04969=1089.841,317.970,-86.406,177.149,22.647,153.451
C04970=1089.846,318.218,-86.438,177.152,22.651,153.452
C04971=1089.852,318.466,-86.470,177.155,22.654,153.452
C04972=1089.857,318.713,-86.502,177.158,22.658,153.452
C04973=1089.863,318.961,-86.534,177.161,22.662,153.453
C04974=1089.869,319.209,-86.565,177.164,22.665,153.453
C04975=1089.874,319.458,-86.598,177.167,22.669,153.454
C04976=1089.880,319.705,-86.631,177.170,22.673,153.454
C04977=1089.886,319.953,-86.662,177.173,22.677,153.454
C04978=1089.892,320.201,-86.694,177.176,22.680,153.455
C04979=1089.897,320.448,-86.726,177.179,22.683,153.455
C04980=1089.903,320.696,-86.759,177.182,22.687,153.456
C04981=1089.909,320.944,-86.791,177.185,22.691,153.456
C04982=1089.914,321.192,-86.823,177.188,22.695,153.456
C04983=1089.920,321.440,-86.855,177.191,22.699,153.457
C04984=1089.926,321.688,-86.888,177.194,22.702,153.457
C04985=1089.931,321.936,-86.920,177.198,22.706,153.458
C04986=1089.937,322.184,-86.952,177.200,22.710,153.458
C04987=1089.943,322.431,-86.985,177.203,22.714,153.459
C04988=1089.949,322.679,-87.016,177.206,22.717,153.459
C04989=1089.954,322.927,-87.050,177.210,22.721,153.459
C04990=1089.960,323.175,-87.082,177.213,22.725,153.460
C04991=1089.966,323.423,-87.114,177.215,22.728,153.460
C04992=1089.972,323.670,-87.146,177.218,22.732,153.461
C04993=1089.977,323.919,-87.179,177.221,22.736,153.461
C04994=1089.983,324.166,-87.212,177.225,22.740,153.461
C04995=1089.989,324.414,-87.244,177.228,22.744,153.462
C04996=1089.994,324.662,-87.277,177.230,22.747,153.462
C04997=1090.000,324.910,-87.309,177.233,22.750,153.463
C04998=1090.007,325.157,-87.341,177.237,22.755,153.463
C04999=1090.012,325.406,-87.374,177.240,22.758,153.463
C05000=1090.018,325.654,-87.407,177.243,22.762,153.464
C05001=1090.024,325.900,-87.439,177.245,22.766,153.464
C05002=1090.030,326.149,-87.471,177.249,22.770,153.465
C05003=1090.035,326.397,-87.504,177.252,22.773,153.465
C05004=1090.041,326.645,-87.536,177.255,22.777,153.466
C05005=1090.047,326.893,-87.570,177.258,22.781,153.466
C05006=1090.053,327.140,-87.602,177.261,22.785,153.467
C05007=1090.059,327.388,-87.634,177.264,22.789,153.467
C05008=1090.064,327.636,-87.668,177.267,22.792,153.467
C05009=1090.070,327.883,-87.700,177.270,22.797,153.468
C05010=1090.077,328.131,-87.733,177.273,22.800,153.468
C05011=1090.082,328.379,-87.766,177.276,22.804,153.469
C05012=1090.088,328.627,-87.798,177.280,22.808,153.469
C05013=1090.094,328.875,-87.832,177.283,22.812,153.470
C05014=1090.100,329.123,-87.864,177.285,22.815,153.470
C05015=1090.106,329.370,-87.896,177.288,22.819,153.471
C05016=1090.115,329.763,-87.949,177.293,22.826,153.471
C05017=1090.124,330.156,-88.001,177.298,22.832,153.472
C05018=1090.134,330.550,-88.053,177.303,22.837,153.473
C05019=1090.143,330.942,-88.105,177.308,22.844,153.473
C05020=1090.149,331.189,-88.138,177.311,22.848,153.474
C05021=1090.155,331.437,-88.171,177.314,22.851,153.474
C05022=1090.161,331.685,-88.204,177.317,22.855,153.475
C05023=1090.167,331.933,-88.238,177.320,22.859,153.475
C05024=1090.173,332.180,-88.270,177.323,22.863,153.476
C05025=1090.179,332.428,-88.304,177.327,22.867,153.476
C05026=1090.184,332.676,-88.337,177.329,22.872,153.477
C05027=1090.190,332.924,-88.370,177.332,22.875,153.477
C05028=1090.196,333.172,-88.403,177.336,22.879,153.478
C05029=1090.201,333.419,-88.436,177.338,22.883,153.478
C05030=1090.207,333.667,-88.469,177.342,22.888,153.479
C05031=1090.213,333.914,-88.502,177.345,22.892,153.479
C05032=1090.218,334.162,-88.535,177.348,22.895,153.480
C05033=1090.224,334.410,-88.569,177.351,22.900,153.480
C05034=1090.230,334.658,-88.603,177.354,22.904,153.481
C05035=1090.236,334.905,-88.636,177.357,22.908,153.481
C05036=1090.242,335.153,-88.669,177.360,22.912,153.482
C05037=1090.247,335.401,-88.702,177.363,22.916,153.482
C05038=1090.253,335.649,-88.736,177.366,22.920,153.483
C05039=1090.258,335.897,-88.769,177.369,22.924,153.483
C05040=1090.265,336.144,-88.802,177.372,22.928,153.484
C05041=1090.270,336.392,-88.836,177.376,22.933,153.484
C05042=1090.277,336.640,-88.869,177.378,22.936,153.485
C05043=1090.282,336.888,-88.903,177.381,22.940,153.485
C05044=1090.288,337.135,-88.937,177.385,22.945,153.486
C05045=1090.294,337.383,-88.970,177.387,22.949,153.486
C05046=1090.300,337.630,-89.004,177.391,22.953,153.487
C05047=1090.306,337.878,-89.037,177.394,22.957,153.487
C05048=1090.311,338.126,-89.070,177.396,22.961,153.488
C05049=1090.317,338.373,-89.104,177.400,22.965,153.488
C05050=1090.323,338.621,-89.138,177.403,22.969,153.489
C05051=1090.328,338.869,-89.171,177.406,22.974,153.489
C05052=1090.334,339.116,-89.205,177.409,22.978,153.490
C05053=1090.340,339.364,-89.238,177.412,22.982,153.491
C05054=1090.346,339.612,-89.273,177.415,22.986,153.491
C05055=1090.352,339.860,-89.306,177.418,22.990,153.492
C05056=1090.358,340.108,-89.340,177.421,22.995,153.492
C05057=1090.363,340.355,-89.374,177.424,22.999,153.493
C05058=1090.369,340.603,-89.408,177.428,23.004,153.493
C05059=1090.375,340.851,-89.441,177.430,23.007,153.494
C05060=1090.380,341.098,-89.475,177.433,23.012,153.494
C05061=1090.386,341.345,-89.509,177.437,23.016,153.495
C05062=1090.392,341.594,-89.543,177.439,23.020,153.496
C05063=1090.398,341.841,-89.577,177.443,23.025,153.496
C05064=1090.404,342.089,-89.610,177.445,23.029,153.497
C05065=1090.410,342.336,-89.644,177.449,23.034,153.497
C05066=1090.416,342.584,-89.678,177.452,23.038,153.498
C05067=1090.421,342.831,-89.712,177.455,23.042,153.498
C05068=1090.431,343.219,-89.765,177.460,23.049,153.499
C05069=1090.440,343.606,-89.818,177.465,23.056,153.500
C05070=1090.449,343.993,-89.871,177.470,23.062,153.501
C05071=1090.458,344.380,-89.924,177.474,23.069,153.502
C05072=1090.464,344.627,-89.958,177.477,23.073,153.503
C05073=1090.470,344.875,-89.993,177.480,23.078,153.503
C05074=1090.475,345.123,-90.027,177.483,23.082,153.504
C05075=1090.481,345.370,-90.061,177.486,23.087,153.504
C05076=1090.487,345.617,-90.095,177.489,23.091,153.505
C05077=1090.493,345.866,-90.129,177.492,23.095,153.506
C05078=1090.498,346.113,-90.164,177.495,23.100,153.506
C05079=1090.504,346.361,-90.198,177.498,23.104,153.507
C05080=1090.510,346.608,-90.232,177.502,23.109,153.507
C05081=1090.517,346.856,-90.266,177.504,23.113,153.508
C05082=1090.522,347.103,-90.301,177.508,23.118,153.509
C05083=1090.528,347.351,-90.335,177.511,23.123,153.509
C05084=1090.534,347.598,-90.369,177.514,23.127,153.510
C05085=1090.539,347.846,-90.404,177.517,23.132,153.510
C05086=1090.545,348.094,-90.438,177.520,23.136,153.511
C05087=1090.551,348.341,-90.472,177.523,23.141,153.512
C05088=1090.557,348.589,-90.507,177.526,23.145,153.512
C05089=1090.563,348.836,-90.541,177.529,23.150,153.513
C05090=1090.569,349.083,-90.576,177.532,23.154,153.514
C05091=1090.574,349.331,-90.611,177.535,23.159,153.514
C05092=1090.580,349.579,-90.645,177.538,23.163,153.515
C05093=1090.586,349.826,-90.679,177.542,23.168,153.516
C05094=1090.592,350.074,-90.714,177.544,23.172,153.516
C05095=1090.598,350.322,-90.748,177.548,23.177,153.517
C05096=1090.603,350.569,-90.784,177.550,23.181,153.517
C05097=1090.610,350.817,-90.818,177.554,23.186,153.518
C05098=1090.615,351.064,-90.853,177.557,23.191,153.519
C05099=1090.621,351.311,-90.887,177.560,23.195,153.519
C05100=1090.627,351.559,-90.922,177.563,23.200,153.520
C05101=1090.633,351.806,-90.956,177.566,23.205,153.521
C05102=1090.639,352.054,-90.991,177.569,23.210,153.521
C05103=1090.644,352.301,-91.026,177.572,23.214,153.522
C05104=1090.651,352.549,-91.061,177.575,23.219,153.523
C05105=1090.656,352.797,-91.095,177.579,23.224,153.523
C05106=1090.662,353.044,-91.130,177.581,23.228,153.524
C05107=1090.668,353.292,-91.165,177.585,23.233,153.525
C05108=1090.674,353.539,-91.200,177.587,23.237,153.525
C05109=1090.680,353.787,-91.235,177.591,23.242,153.526
C05110=1090.686,354.034,-91.269,177.594,23.247,153.527
C05111=1090.692,354.282,-91.305,177.596,23.252,153.528
C05112=1090.697,354.529,-91.339,177.600,23.257,153.528
C05113=1090.703,354.776,-91.374,177.602,23.262,153.529
C05114=1090.709,355.024,-91.409,177.606,23.267,153.530
C05115=1090.714,355.271,-91.444,177.609,23.271,153.530
C05116=1090.721,355.519,-91.480,177.612,23.276,153.531
C05117=1090.726,355.766,-91.514,177.615,23.281,153.532
C05118=1090.732,356.014,-91.550,177.619,23.286,153.532
C05119=1090.738,356.261,-91.584,177.621,23.290,153.533
C05120=1090.747,356.651,-91.639,177.626,23.298,153.534
C05121=1090.756,357.040,-91.695,177.631,23.306,153.535
C05122=1090.765,357.431,-91.751,177.636,23.314,153.536
C05123=1090.775,357.820,-91.806,177.640,23.321,153.538
C05124=1090.781,358.067,-91.841,177.644,23.326,153.538
C05125=1090.787,358.314,-91.877,177.647,23.331,153.539
C05126=1090.793,358.563,-91.912,177.649,23.336,153.540
C05127=1090.798,358.810,-91.947,177.653,23.341,153.541
C05128=1090.805,359.057,-91.982,177.656,23.346,153.541
C05129=1090.810,359.304,-92.017,177.659,23.351,153.542
C05130=1090.816,359.552,-92.053,177.662,23.356,153.543
C05131=1090.822,359.799,-92.089,177.665,23.361,153.544
C05132=1090.828,360.047,-92.123,177.668,23.366,153.544
C05133=1090.834,360.294,-92.159,177.671,23.371,153.545
C05134=1090.840,360.541,-92.194,177.674,23.376,153.546
C05135=1090.846,360.789,-92.230,177.677,23.381,153.547
C05136=1090.851,361.036,-92.265,177.680,23.386,153.547
C05137=1090.857,361.284,-92.301,177.684,23.391,153.548
C05138=1090.863,361.531,-92.337,177.686,23.396,153.549
C05139=1090.869,361.778,-92.372,177.689,23.401,153.550
C05140=1090.875,362.026,-92.408,177.693,23.407,153.551
C05141=1090.880,362.273,-92.443,177.696,23.412,153.551
C05142=1090.887,362.520,-92.478,177.698,23.417,153.552
C05143=1090.893,362.768,-92.514,177.702,23.422,153.553
C05144=1090.899,363.014,-92.550,177.705,23.427,153.554
C05145=1090.905,363.262,-92.586,177.707,23.432,153.554
C05146=1090.911,363.510,-92.621,177.711,23.437,153.555
C05147=1090.917,363.757,-92.657,177.714,23.443,153.556
C05148=1090.922,364.004,-92.693,177.717,23.448,153.557
C05149=1090.928,364.252,-92.728,177.720,23.453,153.558
C05150=1090.935,364.499,-92.765,177.723,23.458,153.558
C05151=1090.940,364.746,-92.800,177.726,23.464,153.559
C05152=1090.946,364.994,-92.836,177.729,23.469,153.560
C05153=1090.952,365.241,-92.872,177.732,23.473,153.561
C05154=1090.958,365.488,-92.908,177.735,23.479,153.562
C05155=1090.964,365.735,-92.943,177.739,23.484,153.562
C05156=1090.970,365.983,-92.979,177.741,23.489,153.563
C05157=1090.975,366.230,-93.016,177.744,23.495,153.564
C05158=1090.981,366.477,-93.051,177.748,23.500,153.565
C05159=1090.987,366.725,-93.087,177.751,23.506,153.566
C05160=1090.993,366.972,-93.124,177.754,23.511,153.567
C05161=1090.999,367.219,-93.159,177.756,23.517,153.568
C05162=1091.004,367.466,-93.196,177.760,23.522,153.569
C05163=1091.010,367.714,-93.232,177.763,23.527,153.569
C05164=1091.016,367.962,-93.267,177.766,23.533,153.570
C05165=1091.022,368.208,-93.304,177.769,23.538,153.571
C05166=1091.028,368.456,-93.339,177.772,23.543,153.572
C05167=1091.034,368.703,-93.376,177.775,23.549,153.573
C05168=1091.040,368.951,-93.412,177.778,23.555,153.574
C05169=1091.045,369.197,-93.448,177.781,23.560,153.575
C05170=1091.052,369.444,-93.485,177.784,23.566,153.576
C05171=1091.057,369.692,-93.521,177.787,23.571,153.576
C05172=1091.067,370.097,-93.581,177.792,23.580,153.578
C05173=1091.077,370.502,-93.640,177.797,23.589,153.579
C05174=1091.086,370.908,-93.699,177.802,23.598,153.581
C05175=1091.096,371.312,-93.759,177.807,23.607,153.582
C05176=1091.103,371.559,-93.796,177.811,23.613,153.583
C05177=1091.108,371.807,-93.831,177.813,23.618,153.584
C05178=1091.114,372.054,-93.868,177.816,23.624,153.585
C05179=1091.120,372.301,-93.904,177.819,23.630,153.586
C05180=1091.126,372.548,-93.941,177.822,23.635,153.587
C05181=1091.132,372.796,-93.977,177.826,23.641,153.588
C05182=1091.138,373.043,-94.014,177.829,23.646,153.589
C05183=1091.144,373.290,-94.051,177.832,23.652,153.590
C05184=1091.150,373.537,-94.087,177.834,23.658,153.591
C05185=1091.156,373.784,-94.124,177.838,23.663,153.591
C05186=1091.162,374.032,-94.161,177.841,23.669,153.592
C05187=1091.168,374.279,-94.197,177.844,23.675,153.593
C05188=1091.174,374.526,-94.234,177.847,23.681,153.594
C05189=1091.180,374.772,-94.270,177.850,23.687,153.595
C05190=1091.185,375.020,-94.307,177.853,23.693,153.596
C05191=1091.192,375.267,-94.344,177.856,23.698,153.597
C05192=1091.197,375.514,-94.381,177.859,23.704,153.598
C05193=1091.203,375.762,-94.418,177.862,23.710,153.599
C05194=1091.209,376.009,-94.454,177.865,23.716,153.600
C05195=1091.215,376.256,-94.491,177.868,23.721,153.601
C05196=1091.221,376.503,-94.528,177.871,23.728,153.602
C05197=1091.227,376.750,-94.565,177.874,23.734,153.603
C05198=1091.232,376.998,-94.602,177.877,23.739,153.604
C05199=1091.239,377.244,-94.639,177.880,23.745,153.605
C05200=1091.245,377.492,-94.676,177.883,23.751,153.606
C05201=1091.251,377.739,-94.712,177.886,23.758,153.607
C05202=1091.256,377.986,-94.749,177.890,23.763,153.608
C05203=1091.262,378.233,-94.786,177.893,23.769,153.609
C05204=1091.269,378.480,-94.824,177.895,23.775,153.610
C05205=1091.274,378.727,-94.861,177.898,23.781,153.611
C05206=1091.280,378.974,-94.898,177.901,23.787,153.612
C05207=1091.287,379.221,-94.935,177.904,23.793,153.613
C05208=1091.292,379.468,-94.972,177.907,23.799,153.614
C05209=1091.298,379.716,-95.009,177.910,23.805,153.615
C05210=1091.304,379.962,-95.046,177.913,23.811,153.616
C05211=1091.310,380.209,-95.083,177.916,23.817,153.617
C05212=1091.316,380.456,-95.121,177.919,23.824,153.619
C05213=1091.321,380.704,-95.158,177.923,23.830,153.620
C05214=1091.328,380.951,-95.195,177.926,23.836,153.621
C05215=1091.334,381.198,-95.232,177.929,23.842,153.622
C05216=1091.340,381.445,-95.270,177.932,23.848,153.623
C05217=1091.347,381.692,-95.307,177.935,23.854,153.624
C05218=1091.352,381.939,-95.344,177.938,23.861,153.625
C05219=1091.358,382.186,-95.381,177.941,23.867,153.626
C05220=1091.364,382.433,-95.419,177.944,23.873,153.627
C05221=1091.371,382.680,-95.456,177.947,23.879,153.628
C05222=1091.377,382.927,-95.494,177.950,23.885,153.629
C05223=1091.382,383.175,-95.531,177.953,23.892,153.630
C05224=1091.388,383.390,-95.564,177.955,23.897,153.631
C05225=1091.393,383.607,-95.597,177.958,23.903,153.632
C05226=1091.398,383.823,-95.630,177.961,23.908,153.633
C05227=1091.403,384.039,-95.662,177.964,23.914,153.634
C05228=1091.408,384.256,-95.695,177.966,23.920,153.635
C05229=1091.413,384.472,-95.729,177.969,23.925,153.636
C05230=1091.418,384.689,-95.762,177.972,23.931,153.637
C05231=1091.424,384.905,-95.795,177.974,23.936,153.638
C05232=1091.429,385.152,-95.832,177.977,23.943,153.639
C05233=1091.435,385.399,-95.870,177.981,23.950,153.641
C05234=1091.442,385.646,-95.908,177.984,23.956,153.642
C05235=1091.448,385.893,-95.946,177.987,23.963,153.643
C05236=1091.453,386.140,-95.983,177.990,23.969,153.644
C05237=1091.459,386.387,-96.021,177.992,23.976,153.645
C05238=1091.465,386.633,-96.059,177.995,23.982,153.646
C05239=1091.471,386.881,-96.096,177.998,23.989,153.648
C05240=1091.477,387.128,-96.134,178.001,23.995,153.649
C05241=1091.483,387.375,-96.172,178.004,24.002,153.650
C05242=1091.489,387.622,-96.210,178.007,24.008,153.651
C05243=1091.496,387.869,-96.248,178.010,24.015,153.652
C05244=1091.502,388.116,-96.285,178.014,24.022,153.654
C05245=1091.507,388.362,-96.323,178.017,24.028,153.655
C05246=1091.514,388.609,-96.362,178.020,24.035,153.656
C05247=1091.520,388.856,-96.400,178.023,24.042,153.657
C05248=1091.526,389.103,-96.438,178.026,24.048,153.658
C05249=1091.531,389.350,-96.476,178.028,24.055,153.660
C05250=1091.538,389.597,-96.514,178.032,24.061,153.661
C05251=1091.544,389.844,-96.552,178.034,24.068,153.662
C05252=1091.550,390.091,-96.590,178.038,24.075,153.663
C05253=1091.556,390.338,-96.628,178.041,24.082,153.664
C05254=1091.562,390.584,-96.666,178.044,24.089,153.666
C05255=1091.569,390.832,-96.704,178.047,24.096,153.667
C05256=1091.574,391.079,-96.743,178.050,24.102,153.668
C05257=1091.580,391.325,-96.781,178.053,24.109,153.669
C05258=1091.587,391.572,-96.819,178.056,24.117,153.671
C05259=1091.593,391.819,-96.857,178.059,24.123,153.672
C05260=1091.599,392.067,-96.895,178.062,24.130,153.673
C05261=1091.605,392.313,-96.934,178.065,24.137,153.674
C05262=1091.611,392.560,-96.972,178.068,24.144,153.676
C05263=1091.617,392.807,-97.011,178.071,24.151,153.677
C05264=1091.622,393.054,-97.049,178.074,24.158,153.678
C05265=1091.629,393.301,-97.087,178.077,24.165,153.680
C05266=1091.635,393.547,-97.126,178.080,24.172,153.681
C05267=1091.641,393.795,-97.164,178.083,24.179,153.682
C05268=1091.647,394.041,-97.203,178.086,24.186,153.684
C05269=1091.654,394.289,-97.241,178.089,24.194,153.685
C05270=1091.659,394.535,-97.280,178.092,24.200,153.686
C05271=1091.666,394.782,-97.318,178.095,24.207,153.688
C05272=1091.671,395.029,-97.357,178.098,24.215,153.689
C05273=1091.678,395.276,-97.396,178.101,24.222,153.690
C05274=1091.683,395.523,-97.434,178.104,24.229,153.692
C05275=1091.690,395.770,-97.473,178.107,24.236,153.693
C05276=1091.695,396.017,-97.512,178.110,24.244,153.694
C05277=1091.702,396.263,-97.550,178.113,24.251,153.696
C05278=1091.707,396.510,-97.590,178.116,24.258,153.697
C05279=1091.714,396.757,-97.628,178.119,24.266,153.698
C05280=1091.720,396.980,-97.663,178.122,24.272,153.700
C05281=1091.725,397.203,-97.698,178.125,24.279,153.701
C05282=1091.730,397.426,-97.733,178.127,24.285,153.702
C05283=1091.736,397.649,-97.768,178.130,24.292,153.703
C05284=1091.741,397.872,-97.803,178.133,24.299,153.705
C05285=1091.747,398.095,-97.838,178.136,24.306,153.706
C05286=1091.752,398.318,-97.874,178.138,24.312,153.707
C05287=1091.758,398.541,-97.909,178.141,24.319,153.709
C05288=1091.763,398.787,-97.948,178.144,24.327,153.710
C05289=1091.770,399.034,-97.987,178.147,24.334,153.711
C05290=1091.776,399.282,-98.026,178.150,24.341,153.713
C05291=1091.781,399.528,-98.065,178.153,24.349,153.714
C05292=1091.788,399.775,-98.104,178.156,24.357,153.716
C05293=1091.794,400.022,-98.143,178.159,24.364,153.717
C05294=1091.800,400.269,-98.182,178.162,24.372,153.719
C05295=1091.807,400.515,-98.221,178.165,24.379,153.720
C05296=1091.813,400.762,-98.261,178.168,24.387,153.722
C05297=1091.818,401.009,-98.300,178.171,24.395,153.723
C05298=1091.824,401.256,-98.339,178.174,24.402,153.725
C05299=1091.830,401.503,-98.379,178.176,24.410,153.726
C05300=1091.837,401.749,-98.418,178.180,24.418,153.728
C05301=1091.843,401.996,-98.457,178.183,24.426,153.729
C05302=1091.849,402.243,-98.497,178.186,24.434,153.731
C05303=1091.855,402.490,-98.536,178.189,24.442,153.732
C05304=1091.861,402.737,-98.575,178.191,24.449,153.734
C05305=1091.867,402.983,-98.614,178.195,24.457,153.735
C05306=1091.874,403.230,-98.654,178.198,24.465,153.737
C05307=1091.880,403.477,-98.693,178.201,24.473,153.738
C05308=1091.886,403.724,-98.733,178.204,24.481,153.740
C05309=1091.892,403.971,-98.772,178.207,24.489,153.741
C05310=1091.898,404.217,-98.812,178.210,24.497,153.743
C05311=1091.904,404.464,-98.852,178.212,24.505,153.745
C05312=1091.910,404.711,-98.891,178.216,24.513,153.746
C05313=1091.916,404.958,-98.931,178.219,24.521,153.748
C05314=1091.922,405.205,-98.971,178.222,24.529,153.749
C05315=1091.929,405.452,-99.011,178.225,24.537,153.751
C05316=1091.934,405.698,-99.050,178.228,24.545,153.752
C05317=1091.941,405.944,-99.090,178.231,24.553,153.754
C05318=1091.947,406.192,-99.129,178.234,24.562,153.756
C05319=1091.953,406.438,-99.170,178.237,24.570,153.757
C05320=1091.959,406.685,-99.209,178.240,24.578,153.759
C05321=1091.965,406.932,-99.249,178.243,24.586,153.760
C05322=1091.972,407.179,-99.289,178.246,24.595,153.762
C05323=1091.978,407.425,-99.329,178.249,24.603,153.764
C05324=1091.983,407.672,-99.368,178.252,24.611,153.765
C05325=1091.990,407.918,-99.408,178.256,24.620,153.767
C05326=1091.996,408.165,-99.448,178.258,24.628,153.769
C05327=1092.001,408.412,-99.488,178.261,24.637,153.770
C05328=1092.008,408.659,-99.528,178.264,24.645,153.772
C05329=1092.014,408.905,-99.568,178.267,24.654,153.774
C05330=1092.021,409.152,-99.608,178.271,24.663,153.776
C05331=1092.026,409.399,-99.649,178.273,24.671,153.777
C05332=1092.032,409.646,-99.689,178.277,24.679,153.779
C05333=1092.039,409.892,-99.729,178.279,24.688,153.781
C05334=1092.045,410.139,-99.769,178.282,24.697,153.782
C05335=1092.051,410.386,-99.810,178.286,24.706,153.784
C05336=1092.056,410.610,-99.846,178.288,24.713,153.786
C05337=1092.062,410.832,-99.882,178.291,24.721,153.787
C05338=1092.068,411.056,-99.919,178.294,24.729,153.789
C05339=1092.073,411.280,-99.955,178.296,24.737,153.790
C05340=1092.079,411.502,-99.991,178.299,24.745,153.792
C05341=1092.085,411.726,-100.028,178.303,24.753,153.794
C05342=1092.090,411.949,-100.064,178.305,24.761,153.795
C05343=1092.096,412.173,-100.101,178.308,24.769,153.797
C05344=1092.102,412.420,-100.142,178.311,24.778,153.799
C05345=1092.108,412.666,-100.182,178.314,24.786,153.800
C05346=1092.115,412.913,-100.222,178.317,24.795,153.802
C05347=1092.120,413.159,-100.263,178.320,24.804,153.804
C05348=1092.127,413.405,-100.304,178.323,24.813,153.806
C05349=1092.133,413.652,-100.344,178.326,24.822,153.808
C05350=1092.139,413.899,-100.385,178.329,24.831,153.810
C05351=1092.145,414.145,-100.425,178.333,24.840,153.811
C05352=1092.152,414.393,-100.466,178.335,24.849,153.813
C05353=1092.158,414.639,-100.507,178.338,24.858,153.815
C05354=1092.165,414.885,-100.547,178.341,24.868,153.817
C05355=1092.170,415.132,-100.588,178.345,24.877,153.819
C05356=1092.177,415.378,-100.628,178.348,24.886,153.821
C05357=1092.183,415.625,-100.670,178.350,24.895,153.823
C05358=1092.190,415.872,-100.710,178.354,24.904,153.824
C05359=1092.196,416.118,-100.751,178.357,24.914,153.826
C05360=1092.202,416.365,-100.791,178.360,24.923,153.828
C05361=1092.208,416.611,-100.833,178.363,24.932,153.830
C05362=1092.215,416.858,-100.873,178.367,24.942,153.832
C05363=1092.220,417.105,-100.914,178.369,24.951,153.834
C05364=1092.226,417.351,-100.955,178.372,24.960,153.836
C05365=1092.233,417.597,-100.996,178.375,24.970,153.838
C05366=1092.239,417.845,-101.037,178.379,24.979,153.840
C05367=1092.246,418.090,-101.078,178.382,24.989,153.842
C05368=1092.252,418.337,-101.119,178.385,24.999,153.844
C05369=1092.258,418.583,-101.161,178.388,25.008,153.846
C05370=1092.264,418.830,-101.202,178.391,25.018,153.848
C05371=1092.271,419.077,-101.242,178.395,25.027,153.850
C05372=1092.276,419.323,-101.284,178.398,25.038,153.852
C05373=1092.282,419.569,-101.325,178.401,25.047,153.854
C05374=1092.290,419.816,-101.367,178.403,25.056,153.856
C05375=1092.295,420.063,-101.407,178.406,25.066,153.858
C05376=1092.301,420.309,-101.449,178.409,25.076,153.860
C05377=1092.308,420.556,-101.491,178.412,25.086,153.862
C05378=1092.315,420.802,-101.532,178.416,25.096,153.864
C05379=1092.321,421.048,-101.573,178.419,25.106,153.866
C05380=1092.327,421.295,-101.615,178.422,25.116,153.868
C05381=1092.333,421.541,-101.656,178.425,25.126,153.870
C05382=1092.340,421.788,-101.697,178.428,25.135,153.872
C05383=1092.346,422.034,-101.739,178.431,25.145,153.874
C05384=1092.352,422.280,-101.780,178.434,25.156,153.877
C05385=1092.359,422.527,-101.822,178.437,25.166,153.879
C05386=1092.365,422.773,-101.864,178.440,25.176,153.881
C05387=1092.371,423.020,-101.905,178.444,25.186,153.883
C05388=1092.377,423.266,-101.947,178.448,25.196,153.885
C05389=1092.383,423.512,-101.988,178.451,25.207,153.887
C05390=1092.390,423.759,-102.030,178.454,25.217,153.890
C05391=1092.396,424.006,-102.072,178.457,25.227,153.892
C05392=1092.404,424.301,-102.122,178.460,25.240,153.894
C05393=1092.411,424.596,-102.171,178.464,25.252,153.897
C05394=1092.419,424.891,-102.222,178.468,25.265,153.900
C05395=1092.426,425.186,-102.272,178.471,25.277,153.902
C05396=1092.433,425.431,-102.314,178.474,25.287,153.904
C05397=1092.439,425.678,-102.356,178.477,25.298,153.907
C05398=1092.445,425.925,-102.397,178.481,25.309,153.909
C05399=1092.452,426.171,-102.440,178.484,25.320,153.911
C05400=1092.458,426.417,-102.481,178.487,25.330,153.913
C05401=1092.465,426.663,-102.524,178.490,25.341,153.916
C05402=1092.471,426.910,-102.566,178.493,25.351,153.918
C05403=1092.477,427.156,-102.608,178.496,25.362,153.920
C05404=1092.483,427.403,-102.650,178.500,25.373,153.923
C05405=1092.490,427.649,-102.692,178.503,25.384,153.925
C05406=1092.496,427.896,-102.734,178.506,25.395,153.927
C05407=1092.503,428.142,-102.777,178.509,25.406,153.930
C05408=1092.509,428.387,-102.819,178.513,25.416,153.932
C05409=1092.516,428.634,-102.861,178.516,25.427,153.934
C05410=1092.522,428.880,-102.903,178.519,25.438,153.937
C05411=1092.528,429.127,-102.946,178.522,25.449,153.939
C05412=1092.535,429.373,-102.989,178.526,25.461,153.941
C05413=1092.541,429.619,-103.030,178.528,25.472,153.944
C05414=1092.548,429.865,-103.073,178.531,25.483,153.946
C05415=1092.554,430.112,-103.116,178.534,25.494,153.949
C05416=1092.560,430.357,-103.158,178.538,25.505,153.951
C05417=1092.567,430.604,-103.200,178.541,25.517,153.954
C05418=1092.573,430.850,-103.244,178.544,25.528,153.956
C05419=1092.580,431.096,-103.286,178.548,25.540,153.958
C05420=1092.586,431.342,-103.328,178.551,25.551,153.961
C05421=1092.593,431.589,-103.371,178.553,25.562,153.963
C05422=1092.599,431.834,-103.414,178.557,25.574,153.966
C05423=1092.605,432.081,-103.457,178.560,25.585,153.968
C05424=1092.612,432.327,-103.499,178.563,25.597,153.971
C05425=1092.619,432.574,-103.542,178.567,25.608,153.973
C05426=1092.624,432.819,-103.585,178.569,25.620,153.976
C05427=1092.631,433.066,-103.627,178.573,25.632,153.979
C05428=1092.637,433.312,-103.670,178.576,25.643,153.981
C05429=1092.644,433.558,-103.714,178.579,25.655,153.984
C05430=1092.650,433.804,-103.756,178.582,25.667,153.986
C05431=1092.657,434.050,-103.799,178.585,25.679,153.989
C05432=1092.663,434.297,-103.842,178.589,25.691,153.991
C05433=1092.670,434.542,-103.885,178.592,25.703,153.994
C05434=1092.675,434.788,-103.928,178.595,25.715,153.997
C05435=1092.682,435.035,-103.971,178.598,25.727,153.999
C05436=1092.689,435.281,-104.014,178.602,25.739,154.002
C05437=1092.695,435.527,-104.058,178.605,25.751,154.005
C05438=1092.702,435.773,-104.101,178.608,25.763,154.007
C05439=1092.708,436.019,-104.144,178.611,25.775,154.010
C05440=1092.719,436.431,-104.216,178.616,25.796,154.015
C05441=1092.729,436.843,-104.289,178.622,25.817,154.019
C05442=1092.740,437.256,-104.362,178.627,25.837,154.024
C05443=1092.752,437.668,-104.435,178.633,25.858,154.028
C05444=1092.757,437.876,-104.471,178.636,25.869,154.031
C05445=1092.768,438.293,-104.545,178.641,25.890,154.036
C05446=1092.773,438.501,-104.582,178.643,25.901,154.038
C05447=1092.779,438.710,-104.618,178.646,25.912,154.040
C05448=1092.785,438.918,-104.656,178.649,25.922,154.043
C05449=1092.790,439.127,-104.693,178.652,25.933,154.045
